C09107=1133.044,378.604,-85.759,-176.914,11.218,149.474
C09108=1133.047,378.356,-85.722,-176.916,11.216,149.474
C09109=1133.051,378.109,-85.685,-176.919,11.213,149.474
C09110=1133.055,377.862,-85.648,-176.921,11.211,149.474
C09111=1133.058,377.615,-85.611,-176.925,11.209,149.474
C09112=1133.062,377.368,-85.574,-176.927,11.207,149.474
C09113=1133.066,377.120,-85.537,-176.930,11.204,149.475
C09114=1133.070,376.874,-85.500,-176.933,11.202,149.475
C09115=1133.073,376.626,-85.463,-176.936,11.200,149.475
C09116=1133.077,376.413,-85.431,-176.938,11.198,149.475
C09117=1133.080,376.200,-85.399,-176.941,11.196,149.475
C09118=1133.084,375.988,-85.367,-176.943,11.194,149.475
C09119=1133.087,375.775,-85.336,-176.945,11.192,149.475
C09120=1133.090,375.562,-85.303,-176.948,11.190,149.475
C09121=1133.093,375.349,-85.272,-176.950,11.188,149.476
C09122=1133.097,375.136,-85.240,-176.953,11.187,149.476
C09123=1133.099,374.924,-85.208,-176.955,11.185,149.476
C09124=1133.104,374.677,-85.171,-176.959,11.182,149.476
C09125=1133.107,374.429,-85.134,-176.962,11.179,149.476
C09126=1133.111,374.182,-85.097,-176.964,11.178,149.476
C09127=1133.114,373.935,-85.061,-176.967,11.175,149.477
C09128=1133.119,373.688,-85.024,-176.970,11.173,149.477
C09129=1133.123,373.440,-84.987,-176.973,11.171,149.477
C09130=1133.126,373.193,-84.950,-176.976,11.168,149.477
C09131=1133.130,372.946,-84.914,-176.979,11.167,149.477
C09132=1133.134,372.699,-84.877,-176.982,11.164,149.477
C09133=1133.138,372.451,-84.840,-176.985,11.161,149.477
C09134=1133.142,372.204,-84.803,-176.988,11.160,149.478
C09135=1133.145,371.957,-84.767,-176.991,11.157,149.478
C09136=1133.149,371.709,-84.730,-176.994,11.155,149.478
C09137=1133.153,371.462,-84.693,-176.997,11.153,149.478
C09138=1133.156,371.215,-84.657,-177.000,11.150,149.478
C09139=1133.160,370.968,-84.620,-177.003,11.148,149.479
C09140=1133.164,370.720,-84.582,-177.006,11.146,149.479
C09141=1133.167,370.473,-84.546,-177.009,11.143,149.479
C09142=1133.171,370.226,-84.510,-177.013,11.141,149.479
C09143=1133.176,369.978,-84.473,-177.015,11.139,149.479
C09144=1133.179,369.731,-84.437,-177.019,11.137,149.480
C09145=1133.183,369.484,-84.400,-177.022,11.134,149.480
C09146=1133.187,369.237,-84.363,-177.025,11.133,149.480
C09147=1133.190,368.989,-84.327,-177.028,11.130,149.480
C09148=1133.194,368.742,-84.290,-177.031,11.128,149.481
C09149=1133.198,368.495,-84.254,-177.034,11.125,149.481
C09150=1133.202,368.248,-84.217,-177.037,11.124,149.481
C09151=1133.206,368.000,-84.180,-177.040,11.121,149.481
C09152=1133.209,367.753,-84.145,-177.044,11.119,149.481
C09153=1133.214,367.506,-84.108,-177.047,11.116,149.482
C09154=1133.217,367.259,-84.072,-177.050,11.114,149.482
C09155=1133.221,367.011,-84.036,-177.053,11.112,149.482
C09156=1133.225,366.764,-83.999,-177.056,11.109,149.482
C09157=1133.229,366.517,-83.963,-177.060,11.107,149.483
C09158=1133.233,366.268,-83.926,-177.063,11.105,149.483
C09159=1133.236,366.022,-83.890,-177.066,11.102,149.483
C09160=1133.240,365.774,-83.853,-177.070,11.100,149.483
C09161=1133.244,365.527,-83.817,-177.072,11.098,149.483
C09162=1133.248,365.280,-83.781,-177.076,11.096,149.484
C09163=1133.251,365.032,-83.745,-177.079,11.093,149.484
C09164=1133.256,364.785,-83.708,-177.083,11.091,149.484
C09165=1133.259,364.537,-83.673,-177.086,11.088,149.484
C09166=1133.263,364.291,-83.636,-177.089,11.086,149.485
C09167=1133.267,364.043,-83.600,-177.092,11.083,149.485
C09168=1133.270,363.796,-83.564,-177.096,11.081,149.485
C09169=1133.275,363.548,-83.528,-177.099,11.079,149.486
C09170=1133.278,363.301,-83.491,-177.102,11.077,149.486
C09171=1133.282,363.054,-83.456,-177.105,11.075,149.486
C09172=1133.286,362.841,-83.424,-177.109,11.072,149.486
C09173=1133.289,362.627,-83.394,-177.111,11.070,149.486
C09174=1133.292,362.415,-83.362,-177.115,11.068,149.487
C09175=1133.295,362.202,-83.331,-177.117,11.066,149.487
C09176=1133.298,361.989,-83.300,-177.120,11.064,149.487
C09177=1133.301,361.776,-83.269,-177.123,11.062,149.487
C09178=1133.305,361.563,-83.239,-177.126,11.060,149.487
C09179=1133.308,361.350,-83.207,-177.129,11.058,149.488
C09180=1133.312,361.102,-83.171,-177.132,11.055,149.488
C09181=1133.316,360.855,-83.136,-177.136,11.053,149.488
C09182=1133.319,360.608,-83.099,-177.139,11.051,149.489
C09183=1133.324,360.360,-83.063,-177.143,11.048,149.489
C09184=1133.327,360.113,-83.028,-177.146,11.046,149.489
C09185=1133.331,359.866,-82.991,-177.150,11.044,149.489
C09186=1133.336,359.619,-82.956,-177.153,11.041,149.490
C09187=1133.339,359.371,-82.920,-177.156,11.039,149.490
C09188=1133.343,359.124,-82.885,-177.160,11.036,149.490
C09189=1133.347,358.876,-82.849,-177.163,11.034,149.490
C09190=1133.351,358.629,-82.812,-177.167,11.032,149.491
C09191=1133.354,358.382,-82.777,-177.170,11.028,149.491
C09192=1133.358,358.134,-82.741,-177.174,11.026,149.491
C09193=1133.362,357.887,-82.705,-177.177,11.024,149.491
C09194=1133.365,357.639,-82.670,-177.181,11.021,149.492
C09195=1133.370,357.391,-82.634,-177.184,11.019,149.492
C09196=1133.374,357.145,-82.599,-177.188,11.017,149.492
C09197=1133.378,356.897,-82.563,-177.191,11.014,149.493
C09198=1133.381,356.650,-82.527,-177.195,11.011,149.493
C09199=1133.385,356.403,-82.491,-177.199,11.009,149.493
C09200=1133.389,356.155,-82.455,-177.202,11.006,149.493
C09201=1133.393,355.907,-82.420,-177.205,11.004,149.494
C09202=1133.396,355.660,-82.384,-177.210,11.001,149.494
C09203=1133.401,355.413,-82.349,-177.213,10.998,149.494
C09204=1133.404,355.166,-82.313,-177.216,10.996,149.494
C09205=1133.408,354.918,-82.278,-177.220,10.994,149.495
C09206=1133.412,354.670,-82.243,-177.224,10.991,149.495
C09207=1133.416,354.422,-82.207,-177.227,10.988,149.495
C09208=1133.420,354.176,-82.172,-177.231,10.986,149.495
C09209=1133.424,353.928,-82.137,-177.234,10.984,149.496
C09210=1133.428,353.680,-82.100,-177.238,10.980,149.496
C09211=1133.432,353.433,-82.065,-177.242,10.978,149.496
C09212=1133.436,353.186,-82.030,-177.245,10.976,149.497
C09213=1133.440,352.938,-81.994,-177.249,10.972,149.497
C09214=1133.444,352.690,-81.959,-177.253,10.970,149.497
C09215=1133.447,352.443,-81.924,-177.256,10.968,149.497
C09216=1133.451,352.195,-81.888,-177.260,10.965,149.498
C09217=1133.455,351.949,-81.853,-177.263,10.962,149.498
C09218=1133.459,351.700,-81.818,-177.267,10.959,149.498
C09219=1133.463,351.453,-81.783,-177.271,10.957,149.498
C09220=1133.467,351.206,-81.748,-177.275,10.954,149.499
C09221=1133.471,350.958,-81.713,-177.278,10.951,149.499
C09222=1133.475,350.711,-81.677,-177.282,10.949,149.499
C09223=1133.478,350.463,-81.642,-177.286,10.946,149.500
C09224=1133.482,350.216,-81.608,-177.289,10.943,149.500
C09225=1133.486,349.968,-81.572,-177.294,10.940,149.500
C09226=1133.489,349.721,-81.537,-177.297,10.938,149.500
C09227=1133.494,349.473,-81.502,-177.301,10.935,149.501
C09228=1133.497,349.260,-81.472,-177.304,10.933,149.501
C09229=1133.501,349.047,-81.441,-177.307,10.930,149.501
C09230=1133.504,348.835,-81.411,-177.309,10.929,149.501
C09231=1133.508,348.621,-81.382,-177.313,10.926,149.501
C09232=1133.511,348.407,-81.351,-177.315,10.924,149.501
C09233=1133.514,348.195,-81.321,-177.317,10.922,149.502
C09234=1133.518,347.982,-81.291,-177.321,10.920,149.502
C09235=1133.521,347.769,-81.260,-177.323,10.918,149.502
C09236=1133.525,347.521,-81.225,-177.326,10.915,149.502
C09237=1133.529,347.273,-81.191,-177.330,10.913,149.502
C09238=1133.532,347.026,-81.156,-177.333,10.911,149.503
C09239=1133.536,346.778,-81.121,-177.336,10.908,149.503
C09240=1133.541,346.531,-81.086,-177.340,10.906,149.503
C09241=1133.545,346.283,-81.051,-177.343,10.903,149.503
C09242=1133.549,346.036,-81.016,-177.346,10.900,149.503
C09243=1133.552,345.788,-80.982,-177.349,10.898,149.504
C09244=1133.557,345.541,-80.947,-177.353,10.895,149.504
C09245=1133.560,345.293,-80.912,-177.356,10.893,149.504
C09246=1133.564,345.045,-80.877,-177.359,10.891,149.504
C09247=1133.568,344.798,-80.843,-177.362,10.888,149.505
C09248=1133.572,344.551,-80.808,-177.366,10.886,149.505
C09249=1133.576,344.303,-80.773,-177.369,10.883,149.505
C09250=1133.580,344.055,-80.739,-177.372,10.880,149.505
C09251=1133.584,343.808,-80.704,-177.375,10.878,149.505
C09252=1133.588,343.560,-80.669,-177.379,10.875,149.506
C09253=1133.592,343.313,-80.634,-177.382,10.873,149.506
C09254=1133.596,343.065,-80.600,-177.385,10.871,149.506
C09255=1133.600,342.817,-80.565,-177.388,10.868,149.506
C09256=1133.604,342.570,-80.531,-177.391,10.865,149.506
C09257=1133.607,342.323,-80.496,-177.395,10.863,149.507
C09258=1133.612,342.075,-80.461,-177.398,10.860,149.507
C09259=1133.616,341.827,-80.427,-177.401,10.858,149.507
C09260=1133.619,341.580,-80.393,-177.405,10.856,149.507
C09261=1133.623,341.332,-80.358,-177.408,10.853,149.507
C09262=1133.627,341.085,-80.324,-177.411,10.850,149.508
C09263=1133.632,340.837,-80.290,-177.414,10.848,149.508
C09264=1133.636,340.589,-80.255,-177.418,10.845,149.508
C09265=1133.640,340.342,-80.221,-177.421,10.843,149.508
C09266=1133.644,340.094,-80.186,-177.424,10.840,149.508
C09267=1133.647,339.847,-80.152,-177.427,10.838,149.509
C09268=1133.651,339.599,-80.117,-177.430,10.835,149.509
C09269=1133.655,339.352,-80.083,-177.434,10.833,149.509
C09270=1133.659,339.103,-80.049,-177.436,10.831,149.509
C09271=1133.663,338.856,-80.015,-177.440,10.829,149.509
C09272=1133.668,338.609,-79.980,-177.443,10.826,149.510
C09273=1133.672,338.361,-79.945,-177.446,10.823,149.510
C09274=1133.675,338.114,-79.912,-177.449,10.821,149.510
C09275=1133.679,337.866,-79.877,-177.453,10.819,149.510
C09276=1133.683,337.618,-79.843,-177.456,10.816,149.510
C09277=1133.686,337.371,-79.809,-177.459,10.813,149.511
C09278=1133.691,337.123,-79.774,-177.462,10.811,149.511
C09279=1133.695,336.875,-79.741,-177.466,10.808,149.511
C09280=1133.699,336.627,-79.706,-177.469,10.806,149.511
C09281=1133.703,336.380,-79.672,-177.472,10.803,149.512
C09282=1133.707,336.132,-79.637,-177.475,10.801,149.512
C09283=1133.711,335.885,-79.604,-177.478,10.798,149.512
C09284=1133.714,335.672,-79.575,-177.482,10.796,149.512
C09285=1133.718,335.458,-79.545,-177.484,10.794,149.512
C09286=1133.721,335.245,-79.516,-177.487,10.792,149.512
C09287=1133.724,335.032,-79.487,-177.490,10.789,149.512
C09288=1133.728,334.819,-79.458,-177.492,10.788,149.513
C09289=1133.731,334.605,-79.428,-177.495,10.785,149.513
C09290=1133.735,334.392,-79.399,-177.498,10.783,149.513
C09291=1133.738,334.178,-79.370,-177.500,10.781,149.513
C09292=1133.743,333.931,-79.335,-177.504,10.779,149.513
C09293=1133.746,333.683,-79.301,-177.507,10.776,149.514
C09294=1133.750,333.436,-79.268,-177.510,10.774,149.514
C09295=1133.754,333.188,-79.233,-177.513,10.771,149.514
C09296=1133.758,332.940,-79.199,-177.516,10.769,149.514
C09297=1133.762,332.693,-79.166,-177.520,10.766,149.514
C09298=1133.766,332.445,-79.132,-177.523,10.764,149.515
C09299=1133.771,332.197,-79.098,-177.526,10.761,149.515
C09300=1133.774,331.950,-79.064,-177.529,10.758,149.515
C09301=1133.778,331.703,-79.030,-177.533,10.756,149.515
C09302=1133.782,331.454,-78.997,-177.536,10.754,149.515
C09303=1133.786,331.207,-78.962,-177.539,10.751,149.515
C09304=1133.790,330.959,-78.929,-177.542,10.748,149.516
C09305=1133.794,330.712,-78.895,-177.546,10.746,149.516
C09306=1133.798,330.464,-78.862,-177.549,10.743,149.516
C09307=1133.802,330.215,-78.828,-177.552,10.741,149.516
C09308=1133.806,329.968,-78.794,-177.555,10.738,149.517
C09309=1133.810,329.721,-78.761,-177.558,10.736,149.517
C09310=1133.814,329.473,-78.727,-177.562,10.733,149.517
C09311=1133.817,329.225,-78.694,-177.565,10.731,149.517
C09312=1133.822,328.978,-78.659,-177.568,10.728,149.517
C09313=1133.826,328.730,-78.626,-177.571,10.726,149.518
C09314=1133.830,328.482,-78.593,-177.574,10.723,149.518
C09315=1133.834,328.235,-78.559,-177.578,10.720,149.518
C09316=1133.838,327.987,-78.525,-177.581,10.718,149.518
C09317=1133.842,327.739,-78.492,-177.584,10.716,149.518
C09318=1133.846,327.492,-78.458,-177.587,10.713,149.518
C09319=1133.850,327.244,-78.425,-177.590,10.710,149.519
C09320=1133.855,326.996,-78.392,-177.594,10.708,149.519
C09321=1133.858,326.748,-78.358,-177.597,10.705,149.519
C09322=1133.862,326.500,-78.324,-177.600,10.703,149.519
C09323=1133.866,326.253,-78.291,-177.603,10.701,149.520
C09324=1133.870,326.005,-78.258,-177.606,10.699,149.520
C09325=1133.874,325.757,-78.225,-177.609,10.696,149.520
C09326=1133.879,325.509,-78.192,-177.612,10.693,149.520
C09327=1133.882,325.262,-78.158,-177.616,10.691,149.520
C09328=1133.886,325.014,-78.124,-177.619,10.688,149.520
C09329=1133.890,324.766,-78.091,-177.622,10.686,149.521
C09330=1133.894,324.518,-78.058,-177.625,10.683,149.521
C09331=1133.898,324.271,-78.025,-177.628,10.680,149.521
C09332=1133.902,324.023,-77.992,-177.631,10.678,149.521
C09333=1133.907,323.775,-77.958,-177.635,10.676,149.521
C09334=1133.911,323.528,-77.925,-177.638,10.673,149.521
C09335=1133.915,323.280,-77.892,-177.641,10.670,149.522
C09336=1133.918,323.031,-77.859,-177.644,10.668,149.522
C09337=1133.922,322.784,-77.825,-177.647,10.665,149.522
C09338=1133.926,322.537,-77.792,-177.651,10.663,149.522
C09339=1133.930,322.289,-77.759,-177.654,10.660,149.523
C09340=1133.934,322.076,-77.731,-177.656,10.658,149.523
C09341=1133.937,321.862,-77.703,-177.660,10.656,149.523
C09342=1133.940,321.649,-77.673,-177.662,10.654,149.523
C09343=1133.944,321.435,-77.645,-177.665,10.651,149.523
C09344=1133.948,321.222,-77.616,-177.667,10.649,149.523
C09345=1133.951,321.008,-77.588,-177.670,10.647,149.523
C09346=1133.955,320.794,-77.560,-177.673,10.645,149.524
C09347=1133.958,320.582,-77.531,-177.675,10.643,149.524
C09348=1133.962,320.334,-77.498,-177.679,10.641,149.524
C09349=1133.966,320.086,-77.466,-177.682,10.638,149.524
C09350=1133.970,319.838,-77.433,-177.685,10.635,149.524
C09351=1133.974,319.590,-77.399,-177.688,10.633,149.525
C09352=1133.978,319.343,-77.367,-177.692,10.630,149.525
C09353=1133.982,319.095,-77.334,-177.695,10.628,149.525
C09354=1133.986,318.847,-77.301,-177.698,10.625,149.525
C09355=1133.991,318.599,-77.268,-177.701,10.622,149.525
C09356=1133.995,318.351,-77.235,-177.704,10.620,149.526
C09357=1133.998,318.104,-77.202,-177.707,10.618,149.526
C09358=1134.002,317.856,-77.169,-177.710,10.615,149.526
C09359=1134.007,317.608,-77.137,-177.714,10.612,149.526
C09360=1134.011,317.360,-77.104,-177.717,10.610,149.526
C09361=1134.014,317.113,-77.071,-177.720,10.607,149.526
C09362=1134.019,316.864,-77.039,-177.723,10.605,149.527
C09363=1134.023,316.617,-77.005,-177.726,10.603,149.527
C09364=1134.026,316.369,-76.973,-177.729,10.600,149.527
C09365=1134.031,316.121,-76.940,-177.732,10.598,149.527
C09366=1134.035,315.873,-76.907,-177.735,10.595,149.527
C09367=1134.038,315.626,-76.875,-177.738,10.593,149.528
C09368=1134.043,315.377,-76.842,-177.742,10.590,149.528
C09369=1134.047,315.130,-76.809,-177.745,10.587,149.528
C09370=1134.050,314.882,-76.777,-177.748,10.585,149.528
C09371=1134.055,314.634,-76.744,-177.751,10.583,149.528
C09372=1134.059,314.387,-76.711,-177.754,10.580,149.529
C09373=1134.063,314.139,-76.680,-177.758,10.577,149.529
C09374=1134.067,313.891,-76.646,-177.761,10.575,149.529
C09375=1134.072,313.643,-76.614,-177.764,10.572,149.529
C09376=1134.075,313.395,-76.581,-177.767,10.570,149.529
C09377=1134.079,313.147,-76.549,-177.770,10.567,149.529
C09378=1134.083,312.899,-76.517,-177.773,10.564,149.530
C09379=1134.087,312.651,-76.484,-177.776,10.562,149.530
C09380=1134.091,312.403,-76.452,-177.780,10.559,149.530
C09381=1134.096,312.156,-76.419,-177.783,10.557,149.530
C09382=1134.100,311.908,-76.387,-177.786,10.554,149.530
C09383=1134.104,311.660,-76.354,-177.789,10.552,149.531
C09384=1134.108,311.412,-76.322,-177.792,10.550,149.531
C09385=1134.112,311.164,-76.290,-177.795,10.547,149.531
C09386=1134.116,310.916,-76.257,-177.798,10.545,149.531
C09387=1134.120,310.669,-76.225,-177.801,10.542,149.531
C09388=1134.125,310.421,-76.193,-177.805,10.540,149.532
C09389=1134.128,310.173,-76.160,-177.807,10.537,149.532
C09390=1134.132,309.925,-76.128,-177.811,10.534,149.532
C09391=1134.136,309.677,-76.096,-177.814,10.532,149.532
C09392=1134.141,309.429,-76.064,-177.817,10.529,149.532
C09393=1134.145,309.182,-76.031,-177.820,10.527,149.533
C09394=1134.148,308.934,-76.000,-177.823,10.524,149.533
C09395=1134.153,308.685,-75.967,-177.827,10.521,149.533
C09396=1134.156,308.472,-75.940,-177.829,10.519,149.533
C09397=1134.160,308.258,-75.912,-177.832,10.517,149.533
C09398=1134.163,308.045,-75.885,-177.835,10.515,149.533
C09399=1134.167,307.831,-75.856,-177.837,10.513,149.533
C09400=1134.170,307.618,-75.829,-177.840,10.511,149.534
C09401=1134.174,307.404,-75.801,-177.843,10.509,149.534
C09402=1134.177,307.191,-75.774,-177.845,10.506,149.534
C09403=1134.181,306.977,-75.746,-177.848,10.504,149.534
C09404=1134.185,306.729,-75.714,-177.851,10.501,149.534
C09405=1134.189,306.481,-75.681,-177.854,10.499,149.535
C09406=1134.194,306.234,-75.650,-177.857,10.496,149.535
C09407=1134.197,305.985,-75.618,-177.861,10.494,149.535
C09408=1134.202,305.737,-75.586,-177.864,10.491,149.535
C09409=1134.206,305.490,-75.554,-177.867,10.489,149.535
C09410=1134.210,305.242,-75.522,-177.870,10.486,149.535
C09411=1134.214,304.993,-75.490,-177.873,10.483,149.536
C09412=1134.218,304.746,-75.458,-177.877,10.481,149.536
C09413=1134.222,304.498,-75.426,-177.879,10.478,149.536
C09414=1134.227,304.250,-75.394,-177.882,10.477,149.536
C09415=1134.230,304.002,-75.362,-177.885,10.474,149.536
C09416=1134.235,303.754,-75.331,-177.888,10.471,149.537
C09417=1134.238,303.506,-75.299,-177.891,10.469,149.537
C09418=1134.243,303.259,-75.267,-177.895,10.466,149.537
C09419=1134.247,303.010,-75.236,-177.898,10.463,149.537
C09420=1134.251,302.762,-75.204,-177.901,10.461,149.537
C09421=1134.255,302.515,-75.172,-177.904,10.459,149.537
C09422=1134.259,302.267,-75.140,-177.907,10.456,149.538
C09423=1134.264,302.018,-75.108,-177.911,10.453,149.538
C09424=1134.268,301.771,-75.077,-177.914,10.451,149.538
C09425=1134.272,301.522,-75.045,-177.917,10.448,149.538
C09426=1134.276,301.275,-75.014,-177.920,10.445,149.538
C09427=1134.280,301.027,-74.982,-177.923,10.443,149.539
C09428=1134.284,300.778,-74.950,-177.926,10.440,149.539
C09429=1134.289,300.531,-74.918,-177.929,10.438,149.539
C09430=1134.293,300.282,-74.887,-177.932,10.436,149.539
C09431=1134.297,300.035,-74.856,-177.935,10.433,149.539
C09432=1134.301,299.787,-74.824,-177.938,10.431,149.539
C09433=1134.305,299.538,-74.793,-177.941,10.428,149.540
C09434=1134.309,299.291,-74.761,-177.944,10.425,149.540
C09435=1134.313,299.043,-74.729,-177.948,10.423,149.540
C09436=1134.317,298.795,-74.699,-177.950,10.420,149.540
C09437=1134.322,298.547,-74.666,-177.954,10.418,149.540
C09438=1134.326,298.299,-74.635,-177.957,10.415,149.540
C09439=1134.330,298.051,-74.603,-177.960,10.413,149.541
C09440=1134.334,297.803,-74.572,-177.963,10.410,149.541
C09441=1134.338,297.555,-74.541,-177.966,10.407,149.541
C09442=1134.342,297.307,-74.509,-177.969,10.405,149.541
C09443=1134.346,297.059,-74.478,-177.973,10.402,149.541
C09444=1134.350,296.811,-74.446,-177.975,10.400,149.542
C09445=1134.355,296.563,-74.415,-177.978,10.398,149.542
C09446=1134.359,296.315,-74.384,-177.981,10.395,149.542
C09447=1134.363,296.067,-74.352,-177.985,10.393,149.542
C09448=1134.367,295.819,-74.321,-177.987,10.390,149.542
C09449=1134.371,295.571,-74.290,-177.991,10.387,149.542
C09450=1134.375,295.323,-74.259,-177.994,10.385,149.543
C09451=1134.380,295.075,-74.228,-177.997,10.382,149.543
C09452=1134.383,294.862,-74.200,-177.999,10.380,149.543
C09453=1134.386,294.648,-74.173,-178.002,10.377,149.543
C09454=1134.390,294.434,-74.147,-178.005,10.376,149.543
C09455=1134.393,294.220,-74.120,-178.008,10.373,149.543
C09456=1134.397,294.007,-74.093,-178.010,10.371,149.544
C09457=1134.401,293.793,-74.066,-178.013,10.369,149.544
C09458=1134.404,293.579,-74.039,-178.016,10.367,149.544
C09459=1134.408,293.365,-74.013,-178.018,10.365,149.544
C09460=1134.412,293.118,-73.982,-178.022,10.362,149.544
C09461=1134.416,292.869,-73.951,-178.024,10.359,149.544
C09462=1134.421,292.621,-73.920,-178.028,10.357,149.545
C09463=1134.424,292.373,-73.888,-178.031,10.354,149.545
C09464=1134.428,292.125,-73.858,-178.034,10.352,149.545
C09465=1134.433,291.877,-73.827,-178.037,10.349,149.545
C09466=1134.437,291.629,-73.795,-178.040,10.346,149.545
C09467=1134.441,291.381,-73.765,-178.043,10.345,149.546
C09468=1134.445,291.133,-73.733,-178.046,10.342,149.546
C09469=1134.449,290.885,-73.703,-178.049,10.340,149.546
C09470=1134.454,290.637,-73.672,-178.052,10.337,149.546
C09471=1134.457,290.389,-73.641,-178.055,10.334,149.546
C09472=1134.462,290.141,-73.610,-178.058,10.332,149.546
C09473=1134.466,289.892,-73.579,-178.062,10.329,149.547
C09474=1134.470,289.645,-73.549,-178.064,10.326,149.547
C09475=1134.474,289.397,-73.518,-178.068,10.324,149.547
C09476=1134.479,289.148,-73.487,-178.071,10.321,149.547
C09477=1134.482,288.900,-73.457,-178.074,10.319,149.547
C09478=1134.487,288.653,-73.426,-178.077,10.316,149.547
C09479=1134.491,288.404,-73.395,-178.080,10.314,149.548
C09480=1134.496,288.156,-73.364,-178.083,10.312,149.548
C09481=1134.499,287.909,-73.333,-178.086,10.309,149.548
C09482=1134.503,287.660,-73.302,-178.089,10.306,149.548
C09483=1134.508,287.412,-73.271,-178.092,10.304,149.548
C09484=1134.512,287.165,-73.241,-178.095,10.301,149.549
C09485=1134.516,286.916,-73.210,-178.098,10.298,149.549
C09486=1134.521,286.667,-73.180,-178.101,10.296,149.549
C09487=1134.524,286.420,-73.150,-178.104,10.293,149.549
C09488=1134.529,286.171,-73.118,-178.108,10.291,149.549
C09489=1134.532,285.923,-73.088,-178.111,10.288,149.549
C09490=1134.537,285.675,-73.058,-178.114,10.285,149.550
C09491=1134.542,285.428,-73.027,-178.116,10.284,149.550
C09492=1134.545,285.179,-72.996,-178.119,10.281,149.550
C09493=1134.549,284.931,-72.965,-178.123,10.279,149.550
C09494=1134.553,284.684,-72.935,-178.126,10.276,149.550
C09495=1134.558,284.436,-72.905,-178.129,10.273,149.551
C09496=1134.562,284.186,-72.874,-178.132,10.271,149.551
C09497=1134.566,283.939,-72.844,-178.135,10.268,149.551
C09498=1134.571,283.691,-72.813,-178.138,10.265,149.551
C09499=1134.575,283.443,-72.783,-178.141,10.263,149.551
C09500=1134.579,283.194,-72.752,-178.144,10.260,149.551
C09501=1134.583,282.946,-72.722,-178.147,10.257,149.552
C09502=1134.587,282.698,-72.692,-178.150,10.256,149.552
C09503=1134.591,282.451,-72.661,-178.153,10.253,149.552
C09504=1134.596,282.202,-72.631,-178.156,10.251,149.552
C09505=1134.600,281.954,-72.601,-178.159,10.248,149.552
C09506=1134.604,281.706,-72.570,-178.162,10.245,149.552
C09507=1134.608,281.458,-72.540,-178.166,10.243,149.553
C09508=1134.612,281.244,-72.514,-178.168,10.240,149.553
C09509=1134.616,281.030,-72.488,-178.172,10.238,149.553
C09510=1134.619,280.816,-72.462,-178.175,10.235,149.553
C09511=1134.623,280.603,-72.436,-178.178,10.232,149.553
C09512=1134.627,280.388,-72.410,-178.181,10.230,149.554
C09513=1134.630,280.175,-72.385,-178.184,10.227,149.554
C09514=1134.634,279.961,-72.358,-178.188,10.225,149.554
C09515=1134.637,279.746,-72.332,-178.191,10.222,149.554
C09516=1134.642,279.498,-72.302,-178.194,10.220,149.555
C09517=1134.646,279.250,-72.271,-178.198,10.216,149.555
C09518=1134.650,279.003,-72.241,-178.201,10.214,149.555
C09519=1134.654,278.754,-72.212,-178.205,10.211,149.555
C09520=1134.659,278.506,-72.182,-178.208,10.208,149.555
C09521=1134.663,278.258,-72.152,-178.212,10.206,149.556
C09522=1134.667,278.009,-72.122,-178.215,10.202,149.556
C09523=1134.670,277.761,-72.092,-178.219,10.200,149.556
C09524=1134.675,277.513,-72.062,-178.222,10.196,149.556
C09525=1134.679,277.265,-72.031,-178.225,10.194,149.556
C09526=1134.683,277.017,-72.002,-178.228,10.191,149.557
C09527=1134.688,276.768,-71.972,-178.232,10.188,149.557
C09528=1134.692,276.521,-71.942,-178.235,10.185,149.557
C09529=1134.696,276.272,-71.912,-178.239,10.183,149.557
C09530=1134.701,276.024,-71.883,-178.242,10.180,149.557
C09531=1134.704,275.777,-71.853,-178.245,10.176,149.557
C09532=1134.709,275.528,-71.823,-178.249,10.174,149.558
C09533=1134.714,275.280,-71.793,-178.251,10.171,149.558
C09534=1134.717,275.032,-71.763,-178.254,10.168,149.558
C09535=1134.722,274.784,-71.734,-178.258,10.166,149.558
C09536=1134.726,274.536,-71.704,-178.261,10.163,149.558
C09537=1134.731,274.287,-71.674,-178.264,10.160,149.558
C09538=1134.735,274.039,-71.644,-178.267,10.157,149.558
C09539=1134.739,273.791,-71.614,-178.271,10.155,149.559
C09540=1134.743,273.543,-71.585,-178.274,10.152,149.559
C09541=1134.747,273.295,-71.556,-178.276,10.149,149.559
C09542=1134.751,273.046,-71.526,-178.279,10.146,149.559
C09543=1134.756,272.798,-71.497,-178.282,10.144,149.559
C09544=1134.760,272.550,-71.466,-178.285,10.141,149.559
C09545=1134.764,272.302,-71.436,-178.289,10.138,149.560
C09546=1134.769,272.053,-71.407,-178.291,10.136,149.560
C09547=1134.773,271.805,-71.377,-178.294,10.134,149.560
C09548=1134.777,271.557,-71.348,-178.297,10.131,149.560
C09549=1134.781,271.309,-71.319,-178.300,10.128,149.560
C09550=1134.785,271.060,-71.289,-178.303,10.125,149.560
C09551=1134.789,270.812,-71.260,-178.306,10.123,149.560
C09552=1134.794,270.564,-71.230,-178.308,10.121,149.560
C09553=1134.798,270.316,-71.201,-178.311,10.118,149.560
C09554=1134.802,270.067,-71.171,-178.314,10.115,149.561
C09555=1134.806,269.819,-71.142,-178.317,10.112,149.561
C09556=1134.810,269.571,-71.112,-178.319,10.110,149.561
C09557=1134.815,269.323,-71.083,-178.322,10.108,149.561
C09558=1134.819,269.075,-71.054,-178.325,10.105,149.561
C09559=1134.823,268.827,-71.024,-178.327,10.103,149.561
C09560=1134.828,268.578,-70.995,-178.330,10.100,149.561
C09561=1134.832,268.330,-70.966,-178.332,10.098,149.561
C09562=1134.836,268.082,-70.936,-178.335,10.095,149.561
C09563=1134.840,267.833,-70.907,-178.337,10.093,149.561
C09564=1134.844,267.620,-70.882,-178.340,10.091,149.561
C09565=1134.848,267.405,-70.856,-178.342,10.089,149.562
C09566=1134.852,267.191,-70.832,-178.344,10.087,149.562
C09567=1134.855,266.978,-70.806,-178.346,10.085,149.562
C09568=1134.859,266.763,-70.781,-178.348,10.083,149.562
C09569=1134.863,266.549,-70.756,-178.351,10.081,149.562
C09570=1134.866,266.336,-70.731,-178.353,10.079,149.562
C09571=1134.870,266.121,-70.706,-178.355,10.077,149.562
C09572=1134.874,265.873,-70.676,-178.357,10.075,149.562
C09573=1134.879,265.625,-70.647,-178.360,10.071,149.562
C09574=1134.883,265.377,-70.618,-178.362,10.069,149.562
C09575=1134.887,265.128,-70.589,-178.364,10.067,149.562
C09576=1134.891,264.880,-70.560,-178.367,10.065,149.562
C09577=1134.896,264.631,-70.530,-178.370,10.063,149.563
C09578=1134.900,264.384,-70.502,-178.372,10.061,149.563
C09579=1134.904,264.135,-70.473,-178.376,10.058,149.563
C09580=1134.908,263.887,-70.443,-178.381,10.054,149.563
C09581=1134.913,263.639,-70.414,-178.385,10.050,149.563
C09582=1134.917,263.390,-70.385,-178.389,10.047,149.564
C09583=1134.922,263.142,-70.356,-178.393,10.044,149.564
C09584=1134.926,262.894,-70.328,-178.396,10.041,149.564
C09585=1134.930,262.646,-70.299,-178.400,10.037,149.564
C09586=1134.934,262.397,-70.269,-178.404,10.034,149.565
C09587=1134.939,262.149,-70.241,-178.408,10.031,149.565
C09588=1134.942,261.901,-70.212,-178.412,10.028,149.565
C09589=1134.947,261.652,-70.183,-178.416,10.024,149.565
C09590=1134.951,261.404,-70.154,-178.420,10.021,149.566
C09591=1134.956,261.156,-70.125,-178.423,10.018,149.566
C09592=1134.960,260.908,-70.096,-178.427,10.015,149.566
C09593=1134.964,260.659,-70.068,-178.430,10.012,149.566
C09594=1134.969,260.411,-70.039,-178.434,10.009,149.566
C09595=1134.973,260.163,-70.010,-178.437,10.006,149.566
C09596=1134.977,259.914,-69.982,-178.441,10.003,149.567
C09597=1134.981,259.667,-69.953,-178.445,9.999,149.567
C09598=1134.986,259.418,-69.924,-178.448,9.996,149.567
C09599=1134.990,259.169,-69.896,-178.451,9.993,149.567
C09600=1134.994,258.921,-69.867,-178.455,9.990,149.567
C09601=1134.999,258.673,-69.839,-178.458,9.987,149.567
C09602=1135.003,258.424,-69.810,-178.461,9.984,149.568
C09603=1135.007,258.177,-69.781,-178.465,9.981,149.568
C09604=1135.012,257.928,-69.753,-178.468,9.978,149.568
C09605=1135.015,257.679,-69.724,-178.470,9.975,149.568
C09606=1135.020,257.432,-69.695,-178.473,9.972,149.568
C09607=1135.024,257.183,-69.667,-178.477,9.969,149.568
C09608=1135.028,256.934,-69.638,-178.480,9.966,149.568
C09609=1135.033,256.686,-69.611,-178.483,9.963,149.568
C09610=1135.037,256.437,-69.582,-178.486,9.961,149.568
C09611=1135.041,256.190,-69.553,-178.489,9.958,149.569
C09612=1135.046,255.941,-69.525,-178.491,9.955,149.568
C09613=1135.050,255.693,-69.497,-178.490,9.954,149.568
C09614=1135.055,255.444,-69.468,-178.489,9.954,149.568
C09615=1135.058,255.196,-69.440,-178.488,9.954,149.567
C09616=1135.064,254.948,-69.412,-178.487,9.953,149.567
C09617=1135.067,254.700,-69.383,-178.486,9.953,149.567
C09618=1135.071,254.451,-69.354,-178.486,9.951,149.566
C09619=1135.076,254.203,-69.326,-178.486,9.950,149.566
C09620=1135.082,253.851,-69.286,-178.487,9.950,149.566
C09621=1135.089,253.497,-69.246,-178.488,9.947,149.566
C09622=1135.107,252.397,-69.120,-177.589,8.141,148.878
C09623=1135.111,252.177,-69.096,-177.592,8.138,148.879
C09624=1135.115,251.958,-69.071,-177.594,8.136,148.879
C09625=1135.119,251.738,-69.046,-177.597,8.133,148.879
C09626=1135.123,251.489,-69.018,-177.599,8.130,148.879
C09627=1135.128,251.241,-68.991,-177.602,8.127,148.879
C09628=1135.132,250.992,-68.963,-177.605,8.124,148.879
C09629=1135.136,250.744,-68.935,-177.608,8.121,148.879
C09630=1135.141,250.496,-68.908,-177.610,8.118,148.879
C09631=1135.145,250.247,-68.880,-177.614,8.114,148.879
C09632=1135.150,249.998,-68.852,-177.616,8.111,148.879
C09633=1135.154,249.751,-68.825,-177.619,8.108,148.879
C09634=1135.158,249.502,-68.797,-177.622,8.105,148.879
C09635=1135.162,249.254,-68.769,-177.624,8.102,148.879
C09636=1135.166,249.005,-68.741,-177.627,8.099,148.879
C09637=1135.171,248.756,-68.714,-177.630,8.096,148.879
C09638=1135.175,248.509,-68.687,-177.633,8.093,148.879
C09639=1135.180,248.260,-68.659,-177.636,8.091,148.879
C09640=1135.184,248.011,-68.631,-177.638,8.088,148.879
C09641=1135.189,247.763,-68.604,-177.641,8.084,148.879
C09642=1135.193,247.515,-68.576,-177.644,8.082,148.879
C09643=1135.197,247.266,-68.548,-177.647,8.078,148.879
C09644=1135.202,247.017,-68.521,-177.650,8.075,148.879
C09645=1135.206,246.769,-68.494,-177.653,8.072,148.880
C09646=1135.210,246.520,-68.466,-177.655,8.069,148.880
C09647=1135.215,246.272,-68.438,-177.658,8.066,148.880
C09648=1135.219,246.024,-68.411,-177.661,8.063,148.880
C09649=1135.224,245.775,-68.384,-177.664,8.060,148.880
C09650=1135.228,245.527,-68.356,-177.667,8.057,148.880
C09651=1135.233,245.278,-68.329,-177.669,8.054,148.880
C09652=1135.237,245.030,-68.302,-177.672,8.051,148.880
C09653=1135.242,244.781,-68.275,-177.675,8.048,148.880
C09654=1135.245,244.533,-68.247,-177.677,8.045,148.880
C09655=1135.250,244.284,-68.220,-177.680,8.043,148.880
C09656=1135.254,244.036,-68.193,-177.683,8.040,148.880
C09657=1135.259,243.788,-68.166,-177.686,8.037,148.880
C09658=1135.263,243.539,-68.138,-177.689,8.034,148.880
C09659=1135.267,243.290,-68.111,-177.691,8.031,148.880
C09660=1135.272,243.042,-68.084,-177.694,8.028,148.880
C09661=1135.277,242.793,-68.057,-177.698,8.024,148.881
C09662=1135.281,242.545,-68.029,-177.700,8.021,148.881
C09663=1135.284,242.297,-68.002,-177.703,8.018,148.881
C09664=1135.289,242.048,-67.975,-177.706,8.016,148.881
C09665=1135.294,241.800,-67.948,-177.708,8.012,148.881
C09666=1135.298,241.551,-67.921,-177.711,8.009,148.881
C09667=1135.303,241.303,-67.894,-177.714,8.006,148.881
C09668=1135.308,241.054,-67.867,-177.717,8.004,148.881
C09669=1135.311,240.805,-67.840,-177.720,8.001,148.881
C09670=1135.315,240.557,-67.813,-177.722,7.998,148.881
C09671=1135.320,240.308,-67.786,-177.725,7.995,148.881
C09672=1135.325,240.060,-67.759,-177.728,7.992,148.881
C09673=1135.328,239.812,-67.732,-177.731,7.989,148.881
C09674=1135.333,239.564,-67.705,-177.734,7.986,148.881
C09675=1135.338,239.315,-67.678,-177.736,7.983,148.881
C09676=1135.343,239.066,-67.651,-177.739,7.980,148.882
C09677=1135.346,238.817,-67.624,-177.742,7.977,148.882
C09678=1135.351,238.569,-67.597,-177.745,7.975,148.882
C09679=1135.355,238.320,-67.570,-177.748,7.972,148.882
C09680=1135.360,238.072,-67.543,-177.750,7.969,148.882
C09681=1135.364,237.823,-67.517,-177.753,7.966,148.882
C09682=1135.369,237.575,-67.490,-177.756,7.963,148.882
C09683=1135.373,237.326,-67.463,-177.759,7.960,148.882
C09684=1135.377,237.078,-67.436,-177.762,7.957,148.882
C09685=1135.382,236.830,-67.409,-177.764,7.954,148.882
C09686=1135.386,236.581,-67.382,-177.767,7.951,148.882
C09687=1135.391,236.333,-67.356,-177.770,7.948,148.882
C09688=1135.395,236.084,-67.329,-177.773,7.945,148.882
C09689=1135.400,235.836,-67.302,-177.776,7.943,148.883
C09690=1135.404,235.564,-67.273,-177.778,7.940,148.883
C09691=1135.409,235.291,-67.244,-177.782,7.936,148.883
C09692=1135.414,235.019,-67.215,-177.785,7.933,148.883
C09693=1135.419,234.747,-67.185,-177.788,7.930,148.883
C09694=1135.423,234.499,-67.159,-177.790,7.927,148.883
C09695=1135.428,234.250,-67.133,-177.793,7.924,148.883
C09696=1135.432,234.002,-67.106,-177.796,7.921,148.883
C09697=1135.436,233.753,-67.079,-177.799,7.918,148.883
C09698=1135.441,233.505,-67.053,-177.802,7.916,148.883
C09699=1135.445,233.256,-67.026,-177.804,7.913,148.883
C09700=1135.450,233.008,-66.999,-177.807,7.910,148.883
C09701=1135.454,232.759,-66.973,-177.810,7.907,148.884
C09702=1135.459,232.510,-66.946,-177.813,7.904,148.884
C09703=1135.463,232.262,-66.920,-177.816,7.901,148.884
C09704=1135.467,232.013,-66.894,-177.819,7.898,148.884
C09705=1135.472,231.765,-66.867,-177.822,7.896,148.884
C09706=1135.476,231.516,-66.841,-177.824,7.893,148.884
C09707=1135.480,231.268,-66.814,-177.827,7.890,148.884
C09708=1135.485,231.019,-66.789,-177.830,7.887,148.884
C09709=1135.489,230.770,-66.761,-177.833,7.884,148.884
C09710=1135.494,230.522,-66.736,-177.836,7.881,148.885
C09711=1135.499,230.274,-66.709,-177.838,7.878,148.885
C09712=1135.503,230.025,-66.683,-177.841,7.875,148.885
C09713=1135.507,229.777,-66.657,-177.844,7.872,148.885
C09714=1135.512,229.528,-66.630,-177.847,7.869,148.885
C09715=1135.516,229.279,-66.604,-177.850,7.867,148.885
C09716=1135.521,229.030,-66.578,-177.853,7.864,148.885
C09717=1135.525,228.782,-66.551,-177.855,7.861,148.885
C09718=1135.529,228.533,-66.525,-177.858,7.859,148.885
C09719=1135.534,228.284,-66.499,-177.860,7.856,148.885
C09720=1135.538,228.037,-66.473,-177.863,7.853,148.885
C09721=1135.543,227.788,-66.447,-177.866,7.850,148.886
C09722=1135.547,227.539,-66.420,-177.869,7.847,148.886
C09723=1135.551,227.291,-66.394,-177.872,7.844,148.886
C09724=1135.556,227.042,-66.369,-177.875,7.842,148.886
C09725=1135.560,226.793,-66.342,-177.878,7.839,148.886
C09726=1135.565,226.544,-66.316,-177.880,7.836,148.886
C09727=1135.569,226.296,-66.290,-177.883,7.833,148.886
C09728=1135.574,226.048,-66.265,-177.886,7.830,148.886
C09729=1135.578,225.799,-66.238,-177.889,7.827,148.887
C09730=1135.583,225.550,-66.212,-177.892,7.824,148.887
C09731=1135.587,225.301,-66.186,-177.895,7.821,148.887
C09732=1135.592,225.053,-66.160,-177.898,7.819,148.887
C09733=1135.596,224.805,-66.134,-177.900,7.817,148.887
C09734=1135.600,224.556,-66.108,-177.903,7.814,148.887
C09735=1135.605,224.307,-66.082,-177.906,7.811,148.887
C09736=1135.609,224.058,-66.056,-177.908,7.808,148.887
C09737=1135.614,223.810,-66.030,-177.911,7.805,148.888
C09738=1135.619,223.561,-66.005,-177.914,7.802,148.888
C09739=1135.623,223.312,-65.979,-177.917,7.799,148.888
C09740=1135.627,223.064,-65.953,-177.920,7.796,148.888
C09741=1135.632,222.816,-65.927,-177.923,7.794,148.888
C09742=1135.636,222.567,-65.901,-177.926,7.791,148.888
C09743=1135.641,222.318,-65.875,-177.928,7.789,148.888
C09744=1135.645,222.069,-65.849,-177.931,7.786,148.888
C09745=1135.650,221.821,-65.824,-177.934,7.783,148.889
C09746=1135.654,221.572,-65.798,-177.936,7.780,148.889
C09747=1135.658,221.324,-65.772,-177.939,7.777,148.889
C09748=1135.663,221.075,-65.747,-177.942,7.775,148.889
C09749=1135.667,220.827,-65.721,-177.945,7.772,148.889
C09750=1135.672,220.578,-65.696,-177.948,7.769,148.889
C09751=1135.676,220.329,-65.670,-177.951,7.766,148.889
C09752=1135.681,220.081,-65.644,-177.953,7.764,148.889
C09753=1135.686,219.832,-65.618,-177.956,7.761,148.890
C09754=1135.690,219.583,-65.592,-177.959,7.758,148.890
C09755=1135.695,219.335,-65.567,-177.962,7.755,148.890
C09756=1135.699,219.086,-65.542,-177.965,7.752,148.890
C09757=1135.703,218.837,-65.516,-177.968,7.750,148.890
C09758=1135.708,218.589,-65.491,-177.970,7.747,148.890
C09759=1135.713,218.340,-65.465,-177.973,7.744,148.890
C09760=1135.717,218.091,-65.439,-177.976,7.742,148.891
C09761=1135.722,217.843,-65.414,-177.979,7.739,148.891
C09762=1135.726,217.594,-65.388,-177.982,7.736,148.891
C09763=1135.730,217.345,-65.364,-177.984,7.733,148.891
C09764=1135.734,217.097,-65.338,-177.987,7.730,148.891
C09765=1135.739,216.848,-65.313,-177.990,7.728,148.891
C09766=1135.743,216.599,-65.287,-177.993,7.725,148.891
C09767=1135.748,216.351,-65.262,-177.996,7.723,148.892
C09768=1135.752,216.102,-65.236,-177.998,7.720,148.892
C09769=1135.757,215.854,-65.211,-178.001,7.717,148.892
C09770=1135.761,215.605,-65.185,-178.004,7.714,148.892
C09771=1135.766,215.355,-65.160,-178.007,7.712,148.892
C09772=1135.771,215.107,-65.135,-178.010,7.709,148.892
C09773=1135.775,214.859,-65.109,-178.013,7.706,148.892
C09774=1135.779,214.610,-65.085,-178.015,7.704,148.893
C09775=1135.783,214.361,-65.059,-178.018,7.701,148.893
C09776=1135.788,214.113,-65.034,-178.021,7.698,148.893
C09777=1135.793,213.864,-65.009,-178.024,7.695,148.893
C09778=1135.797,213.615,-64.983,-178.027,7.693,148.893
C09779=1135.802,213.366,-64.958,-178.030,7.690,148.893
C09780=1135.806,213.117,-64.933,-178.032,7.688,148.894
C09781=1135.810,212.870,-64.908,-178.035,7.685,148.894
C09782=1135.815,212.620,-64.883,-178.038,7.682,148.894
C09783=1135.820,212.372,-64.857,-178.041,7.679,148.894
C09784=1135.824,212.123,-64.832,-178.044,7.677,148.894
C09785=1135.828,211.875,-64.808,-178.047,7.674,148.894
C09786=1135.833,211.626,-64.783,-178.049,7.672,148.894
C09787=1135.838,211.377,-64.757,-178.052,7.669,148.895
C09788=1135.842,211.128,-64.732,-178.055,7.666,148.895
C09789=1135.846,210.880,-64.707,-178.058,7.663,148.895
C09790=1135.851,210.631,-64.682,-178.061,7.660,148.895
C09791=1135.856,210.382,-64.658,-178.063,7.658,148.895
C09792=1135.860,210.133,-64.632,-178.066,7.656,148.896
C09793=1135.865,209.885,-64.608,-178.069,7.653,148.896
C09794=1135.870,209.614,-64.580,-178.072,7.650,148.896
C09795=1135.875,209.343,-64.553,-178.075,7.647,148.896
C09796=1135.880,209.073,-64.526,-178.078,7.645,148.896
C09797=1135.884,208.802,-64.499,-178.081,7.641,148.896
C09798=1135.889,208.554,-64.474,-178.084,7.639,148.897
C09799=1135.894,208.304,-64.449,-178.087,7.636,148.897
C09800=1135.898,208.056,-64.425,-178.090,7.633,148.897
C09801=1135.903,207.808,-64.399,-178.093,7.631,148.897
C09802=1135.907,207.559,-64.375,-178.095,7.629,148.897
C09803=1135.912,207.310,-64.350,-178.098,7.626,148.897
C09804=1135.916,207.061,-64.325,-178.101,7.623,148.898
C09805=1135.920,206.813,-64.300,-178.104,7.620,148.898
C09806=1135.925,206.563,-64.275,-178.107,7.617,148.898
C09807=1135.929,206.315,-64.251,-178.109,7.615,148.898
C09808=1135.934,206.066,-64.227,-178.112,7.613,148.898
C09809=1135.939,205.817,-64.201,-178.115,7.610,148.898
C09810=1135.943,205.569,-64.177,-178.118,7.607,148.899
C09811=1135.948,205.320,-64.152,-178.121,7.605,148.899
C09812=1135.952,205.071,-64.128,-178.124,7.602,148.899
C09813=1135.957,204.822,-64.103,-178.126,7.599,148.899
C09814=1135.962,204.574,-64.079,-178.130,7.597,148.899
C09815=1135.966,204.324,-64.054,-178.132,7.594,148.900
C09816=1135.970,204.077,-64.029,-178.135,7.592,148.900
C09817=1135.975,203.828,-64.005,-178.138,7.589,148.900
C09818=1135.979,203.579,-63.980,-178.141,7.586,148.900
C09819=1135.984,203.330,-63.955,-178.144,7.584,148.900
C09820=1135.989,203.082,-63.931,-178.146,7.582,148.901
C09821=1135.993,202.832,-63.906,-178.149,7.579,148.901
C09822=1135.998,202.584,-63.882,-178.152,7.576,148.901
C09823=1136.003,202.335,-63.858,-178.155,7.574,148.901
C09824=1136.006,202.086,-63.833,-178.157,7.571,148.901
C09825=1136.012,201.837,-63.808,-178.160,7.569,148.901
C09826=1136.016,201.589,-63.784,-178.163,7.566,148.902
C09827=1136.020,201.340,-63.760,-178.166,7.564,148.902
C09828=1136.025,201.091,-63.735,-178.169,7.561,148.902
C09829=1136.029,200.843,-63.711,-178.172,7.558,148.902
C09830=1136.034,200.594,-63.687,-178.175,7.556,148.902
C09831=1136.039,200.344,-63.663,-178.177,7.554,148.903
C09832=1136.043,200.096,-63.639,-178.180,7.551,148.903
C09833=1136.048,199.847,-63.614,-178.183,7.548,148.903
C09834=1136.052,199.599,-63.590,-178.186,7.545,148.903
C09835=1136.056,199.350,-63.566,-178.188,7.543,148.903
C09836=1136.061,199.101,-63.541,-178.191,7.541,148.904
C09837=1136.066,198.852,-63.517,-178.195,7.538,148.904
C09838=1136.070,198.603,-63.493,-178.197,7.536,148.904
C09839=1136.075,198.354,-63.468,-178.200,7.533,148.904
C09840=1136.079,198.106,-63.444,-178.203,7.530,148.904
C09841=1136.084,197.857,-63.420,-178.205,7.528,148.905
C09842=1136.088,197.609,-63.396,-178.208,7.526,148.905
C09843=1136.094,197.359,-63.372,-178.211,7.523,148.905
C09844=1136.097,197.110,-63.348,-178.214,7.520,148.905
C09845=1136.102,196.862,-63.324,-178.217,7.518,148.905
C09846=1136.106,196.613,-63.300,-178.220,7.515,148.906
C09847=1136.112,196.364,-63.276,-178.223,7.513,148.906
C09848=1136.116,196.116,-63.252,-178.225,7.511,148.906
C09849=1136.120,195.867,-63.227,-178.228,7.508,148.906
C09850=1136.125,195.617,-63.204,-178.231,7.505,148.906
C09851=1136.130,195.369,-63.179,-178.233,7.503,148.907
C09852=1136.134,195.120,-63.156,-178.237,7.501,148.907
C09853=1136.139,194.871,-63.132,-178.239,7.498,148.907
C09854=1136.143,194.623,-63.108,-178.242,7.496,148.907
C09855=1136.148,194.374,-63.084,-178.245,7.493,148.908
C09856=1136.152,194.125,-63.060,-178.248,7.491,148.908
C09857=1136.157,193.875,-63.036,-178.250,7.489,148.908
C09858=1136.161,193.627,-63.012,-178.253,7.486,148.908
C09859=1136.166,193.379,-62.988,-178.257,7.483,148.908
C09860=1136.171,193.130,-62.964,-178.259,7.481,148.909
C09861=1136.175,192.881,-62.940,-178.262,7.479,148.909
C09862=1136.180,192.632,-62.917,-178.265,7.476,148.909
C09863=1136.184,192.384,-62.893,-178.268,7.474,148.909
C09864=1136.189,192.135,-62.869,-178.270,7.471,148.910
C09865=1136.194,191.886,-62.845,-178.274,7.468,148.910
C09866=1136.198,191.636,-62.821,-178.276,7.466,148.910
C09867=1136.203,191.387,-62.798,-178.279,7.464,148.910
C09868=1136.207,191.139,-62.774,-178.282,7.461,148.910
C09869=1136.212,190.890,-62.750,-178.284,7.459,148.911
C09870=1136.216,190.641,-62.726,-178.288,7.456,148.911
C09871=1136.221,190.392,-62.703,-178.290,7.453,148.911
C09872=1136.226,190.143,-62.680,-178.293,7.452,148.911
C09873=1136.230,189.895,-62.655,-178.296,7.449,148.912
C09874=1136.235,189.646,-62.632,-178.299,7.446,148.912
C09875=1136.239,189.397,-62.609,-178.301,7.444,148.912
C09876=1136.244,189.148,-62.585,-178.305,7.442,148.912
C09877=1136.248,188.899,-62.561,-178.308,7.439,148.912
C09878=1136.253,188.650,-62.538,-178.310,7.437,148.913
C09879=1136.258,188.402,-62.514,-178.313,7.434,148.913
C09880=1136.262,188.153,-62.490,-178.316,7.432,148.913
C09881=1136.267,187.904,-62.467,-178.319,7.430,148.913
C09882=1136.272,187.655,-62.444,-178.322,7.427,148.914
C09883=1136.276,187.406,-62.420,-178.324,7.425,148.914
C09884=1136.281,187.157,-62.396,-178.327,7.422,148.914
C09885=1136.285,186.908,-62.373,-178.330,7.420,148.914
C09886=1136.289,186.660,-62.350,-178.333,7.418,148.915
C09887=1136.294,186.411,-62.326,-178.336,7.415,148.915
C09888=1136.298,186.162,-62.303,-178.338,7.413,148.915
C09889=1136.303,185.913,-62.279,-178.341,7.410,148.915
C09890=1136.308,185.664,-62.256,-178.345,7.408,148.916
C09891=1136.313,185.415,-62.233,-178.347,7.406,148.916
C09892=1136.318,185.167,-62.210,-178.350,7.403,148.916
C09893=1136.323,184.918,-62.186,-178.352,7.401,148.916
C09894=1136.327,184.669,-62.164,-178.356,7.399,148.917
C09895=1136.331,184.421,-62.140,-178.358,7.396,148.917
C09896=1136.336,184.172,-62.116,-178.361,7.394,148.917
C09897=1136.340,183.923,-62.093,-178.364,7.391,148.917
C09898=1136.346,183.653,-62.068,-178.367,7.388,148.918
C09899=1136.351,183.383,-62.043,-178.370,7.387,148.918
C09900=1136.355,183.113,-62.018,-178.373,7.384,148.918
C09901=1136.360,182.844,-61.992,-178.376,7.381,148.918
C09902=1136.365,182.595,-61.969,-178.379,7.379,148.919
C09903=1136.369,182.346,-61.945,-178.382,7.377,148.919
C09904=1136.374,182.098,-61.923,-178.385,7.374,148.919
C09905=1136.379,181.849,-61.900,-178.388,7.371,148.919
C09906=1136.383,181.600,-61.876,-178.390,7.370,148.920
C09907=1136.388,181.350,-61.854,-178.393,7.367,148.920
C09908=1136.392,181.101,-61.831,-178.396,7.365,148.920
C09909=1136.397,180.852,-61.808,-178.399,7.362,148.920
C09910=1136.402,180.603,-61.784,-178.401,7.360,148.921
C09911=1136.406,180.355,-61.762,-178.405,7.358,148.921
C09912=1136.411,180.106,-61.738,-178.407,7.355,148.921
C09913=1136.416,179.857,-61.715,-178.410,7.353,148.922
C09914=1136.420,179.608,-61.692,-178.413,7.350,148.922
C09915=1136.425,179.359,-61.670,-178.416,7.349,148.922
C09916=1136.430,179.110,-61.647,-178.419,7.346,148.922
C09917=1136.434,178.862,-61.624,-178.421,7.344,148.923
C09918=1136.439,178.613,-61.601,-178.425,7.341,148.923
C09919=1136.443,178.364,-61.577,-178.427,7.339,148.923
C09920=1136.448,178.114,-61.555,-178.430,7.337,148.923
C09921=1136.453,177.866,-61.532,-178.432,7.335,148.924
C09922=1136.457,177.617,-61.509,-178.436,7.332,148.924
C09923=1136.462,177.368,-61.486,-178.438,7.329,148.924
C09924=1136.467,177.118,-61.463,-178.441,7.328,148.924
C09925=1136.470,176.870,-61.441,-178.444,7.325,148.925
C09926=1136.476,176.621,-61.418,-178.447,7.323,148.925
C09927=1136.480,176.372,-61.396,-178.450,7.321,148.925
C09928=1136.485,176.123,-61.372,-178.452,7.318,148.925
C09929=1136.489,175.874,-61.349,-178.455,7.316,148.926
C09930=1136.494,175.625,-61.327,-178.458,7.314,148.926
C09931=1136.498,175.377,-61.304,-178.461,7.311,148.926
C09932=1136.503,175.128,-61.281,-178.464,7.310,148.927
C09933=1136.508,174.879,-61.259,-178.467,7.307,148.927
C09934=1136.513,174.630,-61.236,-178.469,7.305,148.927
C09935=1136.517,174.381,-61.214,-178.472,7.302,148.927
C09936=1136.522,174.132,-61.191,-178.475,7.300,148.928
C09937=1136.526,173.884,-61.168,-178.478,7.298,148.928
C09938=1136.531,173.634,-61.146,-178.481,7.296,148.928
C09939=1136.535,173.385,-61.123,-178.484,7.293,148.928
C09940=1136.541,173.136,-61.101,-178.486,7.292,148.929
C09941=1136.545,172.887,-61.078,-178.490,7.289,148.929
C09942=1136.550,172.638,-61.055,-178.492,7.287,148.929
C09943=1136.554,172.390,-61.033,-178.495,7.284,148.930
C09944=1136.559,172.140,-61.010,-178.497,7.282,148.930
C09945=1136.563,171.891,-60.987,-178.501,7.280,148.930
C09946=1136.568,171.643,-60.966,-178.503,7.278,148.931
C09947=1136.573,171.393,-60.943,-178.506,7.275,148.931
C09948=1136.577,171.144,-60.920,-178.509,7.273,148.931
C09949=1136.583,170.895,-60.898,-178.512,7.271,148.931
C09950=1136.587,170.647,-60.875,-178.514,7.269,148.932
C09951=1136.591,170.398,-60.854,-178.518,7.266,148.932
C09952=1136.596,170.148,-60.831,-178.520,7.265,148.932
C09953=1136.600,169.900,-60.808,-178.523,7.262,148.932
C09954=1136.605,169.651,-60.786,-178.526,7.260,148.933
C09955=1136.610,169.401,-60.764,-178.529,7.258,148.933
C09956=1136.615,169.153,-60.741,-178.531,7.255,148.933
C09957=1136.619,168.904,-60.719,-178.535,7.253,148.934
C09958=1136.624,168.654,-60.697,-178.537,7.251,148.934
C09959=1136.629,168.406,-60.674,-178.540,7.248,148.934
C09960=1136.633,168.157,-60.652,-178.543,7.247,148.934
C09961=1136.638,167.908,-60.631,-178.546,7.245,148.935
C09962=1136.643,167.659,-60.608,-178.549,7.242,148.935
C09963=1136.647,167.411,-60.586,-178.551,7.240,148.935
C09964=1136.652,167.161,-60.563,-178.555,7.238,148.936
C09965=1136.657,166.912,-60.541,-178.557,7.236,148.936
C09966=1136.662,166.663,-60.519,-178.560,7.233,148.936
C09967=1136.666,166.414,-60.497,-178.563,7.231,148.937
C09968=1136.670,166.166,-60.475,-178.566,7.229,148.937
C09969=1136.675,165.916,-60.452,-178.568,7.227,148.937
C09970=1136.680,165.667,-60.430,-178.572,7.224,148.937
C09971=1136.684,165.418,-60.408,-178.574,7.222,148.938
C09972=1136.689,165.169,-60.387,-178.577,7.221,148.938
C09973=1136.694,164.920,-60.365,-178.580,7.218,148.938
C09974=1136.699,164.671,-60.343,-178.583,7.216,148.939
C09975=1136.704,164.422,-60.320,-178.585,7.213,148.939
C09976=1136.708,164.173,-60.299,-178.588,7.212,148.939
C09977=1136.712,163.924,-60.276,-178.591,7.209,148.940
C09978=1136.717,163.676,-60.254,-178.594,7.207,148.940
C09979=1136.721,163.426,-60.232,-178.596,7.205,148.940
C09980=1136.726,163.178,-60.210,-178.600,7.203,148.940
C09981=1136.731,162.929,-60.188,-178.602,7.201,148.941
C09982=1136.735,162.680,-60.167,-178.605,7.198,148.941
C09983=1136.741,162.431,-60.144,-178.608,7.197,148.941
C09984=1136.745,162.182,-60.122,-178.611,7.194,148.942
C09985=1136.750,161.933,-60.101,-178.613,7.192,148.942
C09986=1136.754,161.684,-60.079,-178.616,7.190,148.942
C09987=1136.759,161.435,-60.057,-178.619,7.188,148.943
C09988=1136.764,161.185,-60.036,-178.622,7.186,148.943
C09989=1136.769,160.936,-60.014,-178.625,7.183,148.943
C09990=1136.774,160.688,-59.992,-178.628,7.181,148.944
C09991=1136.778,160.438,-59.970,-178.630,7.180,148.944
C09992=1136.783,160.190,-59.949,-178.633,7.177,148.944
C09993=1136.787,159.940,-59.926,-178.636,7.175,148.944
C09994=1136.792,159.692,-59.905,-178.639,7.173,148.945
C09995=1136.796,159.442,-59.883,-178.642,7.171,148.945
C09996=1136.801,159.193,-59.862,-178.644,7.169,148.945
//INST
///DATE 2021/06/25 14:32
///ATTR SC,RW,RJ
////FRAME ROBOT
///GROUP1 RB1
NOP
MOVL C00000 V=800.0 PL=0
MOVL C00001 V=800.0 PL=0
MOVL C00002 V=800.0 PL=0
MOVL C00003 V=800.0 PL=0
MOVL C00004 V=800.0 PL=0
MOVL C00005 V=800.0 PL=0
MOVL C00006 V=800.0 PL=0
MOVL C00007 V=800.0 PL=0
MOVL C00008 V=800.0 PL=0
MOVL C00009 V=800.0 PL=0
MOVL C00010 V=800.0 PL=0
MOVL C00011 V=800.0 PL=0
MOVL C00012 V=800.0 PL=0
MOVL C00013 V=800.0 PL=0
MOVL C00014 V=800.0 PL=0
MOVL C00015 V=800.0 PL=0
MOVL C00016 V=800.0 PL=0
MOVL C00017 V=800.0 PL=0
MOVL C00018 V=800.0 PL=0
MOVL C00019 V=800.0 PL=0
MOVL C00020 V=800.0 PL=0
MOVL C00021 V=800.0 PL=0
MOVL C00022 V=800.0 PL=0
MOVL C00023 V=800.0 PL=0
MOVL C00024 V=800.0 PL=0
MOVL C00025 V=800.0 PL=0
MOVL C00026 V=800.0 PL=0
MOVL C00027 V=800.0 PL=0
MOVL C00028 V=800.0 PL=0
MOVL C00029 V=800.0 PL=0
MOVL C00030 V=800.0 PL=0
MOVL C00031 V=800.0 PL=0
MOVL C00032 V=800.0 PL=0
MOVL C00033 V=800.0 PL=0
MOVL C00034 V=800.0 PL=0
MOVL C00035 V=800.0 PL=0
MOVL C00036 V=800.0 PL=0
MOVL C00037 V=800.0 PL=0
MOVL C00038 V=800.0 PL=0
MOVL C00039 V=800.0 PL=0
MOVL C00040 V=800.0 PL=0
MOVL C00041 V=800.0 PL=0
MOVL C00042 V=800.0 PL=0
MOVL C00043 V=800.0 PL=0
MOVL C00044 V=800.0 PL=0
MOVL C00045 V=800.0 PL=0
MOVL C00046 V=800.0 PL=0
MOVL C00047 V=800.0 PL=0
MOVL C00048 V=800.0 PL=0
MOVL C00049 V=800.0 PL=0
MOVL C00050 V=800.0 PL=0
MOVL C00051 V=800.0 PL=0
MOVL C00052 V=800.0 PL=0
MOVL C00053 V=800.0 PL=0
MOVL C00054 V=800.0 PL=0
MOVL C00055 V=800.0 PL=0
MOVL C00056 V=800.0 PL=0
MOVL C00057 V=800.0 PL=0
MOVL C00058 V=800.0 PL=0
MOVL C00059 V=800.0 PL=0
MOVL C00060 V=800.0 PL=0
MOVL C00061 V=800.0 PL=0
MOVL C00062 V=800.0 PL=0
MOVL C00063 V=800.0 PL=0
MOVL C00064 V=800.0 PL=0
MOVL C00065 V=800.0 PL=0
MOVL C00066 V=800.0 PL=0
MOVL C00067 V=800.0 PL=0
MOVL C00068 V=800.0 PL=0
MOVL C00069 V=800.0 PL=0
MOVL C00070 V=800.0 PL=0
MOVL C00071 V=800.0 PL=0
MOVL C00072 V=800.0 PL=0
MOVL C00073 V=800.0 PL=0
MOVL C00074 V=800.0 PL=0
MOVL C00075 V=800.0 PL=0
MOVL C00076 V=800.0 PL=0
MOVL C00077 V=800.0 PL=0
MOVL C00078 V=800.0 PL=0
MOVL C00079 V=800.0 PL=0
MOVL C00080 V=800.0 PL=0
MOVL C00081 V=800.0 PL=0
MOVL C00082 V=800.0 PL=0
MOVL C00083 V=800.0 PL=0
MOVL C00084 V=800.0 PL=0
MOVL C00085 V=800.0 PL=0
MOVL C00086 V=800.0 PL=0
MOVL C00087 V=800.0 PL=0
MOVL C00088 V=800.0 PL=0
MOVL C00089 V=800.0 PL=0
MOVL C00090 V=800.0 PL=0
MOVL C00091 V=800.0 PL=0
MOVL C00092 V=800.0 PL=0
MOVL C00093 V=800.0 PL=0
MOVL C00094 V=800.0 PL=0
MOVL C00095 V=800.0 PL=0
MOVL C00096 V=800.0 PL=0
MOVL C00097 V=800.0 PL=0
MOVL C00098 V=800.0 PL=0
MOVL C00099 V=800.0 PL=0
MOVL C00100 V=800.0 PL=0
MOVL C00101 V=800.0 PL=0
MOVL C00102 V=800.0 PL=0
MOVL C00103 V=800.0 PL=0
MOVL C00104 V=800.0 PL=0
MOVL C00105 V=800.0 PL=0
MOVL C00106 V=800.0 PL=0
MOVL C00107 V=800.0 PL=0
MOVL C00108 V=800.0 PL=0
MOVL C00109 V=800.0 PL=0
MOVL C00110 V=800.0 PL=0
MOVL C00111 V=800.0 PL=0
MOVL C00112 V=800.0 PL=0
MOVL C00113 V=800.0 PL=0
MOVL C00114 V=800.0 PL=0
MOVL C00115 V=800.0 PL=0
MOVL C00116 V=800.0 PL=0
MOVL C00117 V=800.0 PL=0
MOVL C00118 V=800.0 PL=0
MOVL C00119 V=800.0 PL=0
MOVL C00120 V=800.0 PL=0
MOVL C00121 V=800.0 PL=0
MOVL C00122 V=800.0 PL=0
MOVL C00123 V=800.0 PL=0
MOVL C00124 V=800.0 PL=0
MOVL C00125 V=800.0 PL=0
MOVL C00126 V=800.0 PL=0
MOVL C00127 V=800.0 PL=0
MOVL C00128 V=800.0 PL=0
MOVL C00129 V=800.0 PL=0
MOVL C00130 V=800.0 PL=0
MOVL C00131 V=800.0 PL=0
MOVL C00132 V=800.0 PL=0
MOVL C00133 V=800.0 PL=0
MOVL C00134 V=800.0 PL=0
MOVL C00135 V=800.0 PL=0
MOVL C00136 V=800.0 PL=0
MOVL C00137 V=800.0 PL=0
MOVL C00138 V=800.0 PL=0
MOVL C00139 V=800.0 PL=0
MOVL C00140 V=800.0 PL=0
MOVL C00141 V=800.0 PL=0
MOVL C00142 V=800.0 PL=0
MOVL C00143 V=800.0 PL=0
MOVL C00144 V=800.0 PL=0
MOVL C00145 V=800.0 PL=0
MOVL C00146 V=800.0 PL=0
MOVL C00147 V=800.0 PL=0
MOVL C00148 V=800.0 PL=0
MOVL C00149 V=800.0 PL=0
MOVL C00150 V=800.0 PL=0
MOVL C00151 V=800.0 PL=0
MOVL C00152 V=800.0 PL=0
MOVL C00153 V=800.0 PL=0
MOVL C00154 V=800.0 PL=0
MOVL C00155 V=800.0 PL=0
MOVL C00156 V=800.0 PL=0
MOVL C00157 V=800.0 PL=0
MOVL C00158 V=800.0 PL=0
MOVL C00159 V=800.0 PL=0
MOVL C00160 V=800.0 PL=0
MOVL C00161 V=800.0 PL=0
MOVL C00162 V=800.0 PL=0
MOVL C00163 V=800.0 PL=0
MOVL C00164 V=800.0 PL=0
MOVL C00165 V=800.0 PL=0
MOVL C00166 V=800.0 PL=0
MOVL C00167 V=800.0 PL=0
MOVL C00168 V=800.0 PL=0
MOVL C00169 V=800.0 PL=0
MOVL C00170 V=800.0 PL=0
MOVL C00171 V=800.0 PL=0
MOVL C00172 V=800.0 PL=0
MOVL C00173 V=800.0 PL=0
MOVL C00174 V=800.0 PL=0
MOVL C00175 V=800.0 PL=0
MOVL C00176 V=800.0 PL=0
MOVL C00177 V=800.0 PL=0
MOVL C00178 V=800.0 PL=0
MOVL C00179 V=800.0 PL=0
MOVL C00180 V=800.0 PL=0
MOVL C00181 V=800.0 PL=0
MOVL C00182 V=800.0 PL=0
MOVL C00183 V=800.0 PL=0
MOVL C00184 V=800.0 PL=0
MOVL C00185 V=800.0 PL=0
MOVL C00186 V=800.0 PL=0
MOVL C00187 V=800.0 PL=0
MOVL C00188 V=800.0 PL=0
MOVL C00189 V=800.0 PL=0
MOVL C00190 V=800.0 PL=0
MOVL C00191 V=800.0 PL=0
MOVL C00192 V=800.0 PL=0
MOVL C00193 V=800.0 PL=0
MOVL C00194 V=800.0 PL=0
MOVL C00195 V=800.0 PL=0
MOVL C00196 V=800.0 PL=0
MOVL C00197 V=800.0 PL=0
MOVL C00198 V=800.0 PL=0
MOVL C00199 V=800.0 PL=0
MOVL C00200 V=800.0 PL=0
MOVL C00201 V=800.0 PL=0
MOVL C00202 V=800.0 PL=0
MOVL C00203 V=800.0 PL=0
MOVL C00204 V=800.0 PL=0
MOVL C00205 V=800.0 PL=0
MOVL C00206 V=800.0 PL=0
MOVL C00207 V=800.0 PL=0
MOVL C00208 V=800.0 PL=0
MOVL C00209 V=800.0 PL=0
MOVL C00210 V=800.0 PL=0
MOVL C00211 V=800.0 PL=0
MOVL C00212 V=800.0 PL=0
MOVL C00213 V=800.0 PL=0
MOVL C00214 V=800.0 PL=0
MOVL C00215 V=800.0 PL=0
MOVL C00216 V=800.0 PL=0
MOVL C00217 V=800.0 PL=0
MOVL C00218 V=800.0 PL=0
MOVL C00219 V=800.0 PL=0
MOVL C00220 V=800.0 PL=0
MOVL C00221 V=800.0 PL=0
MOVL C00222 V=800.0 PL=0
MOVL C00223 V=800.0 PL=0
MOVL C00224 V=800.0 PL=0
MOVL C00225 V=800.0 PL=0
MOVL C00226 V=800.0 PL=0
MOVL C00227 V=800.0 PL=0
MOVL C00228 V=800.0 PL=0
MOVL C00229 V=800.0 PL=0
MOVL C00230 V=800.0 PL=0
MOVL C00231 V=800.0 PL=0
MOVL C00232 V=800.0 PL=0
MOVL C00233 V=800.0 PL=0
MOVL C00234 V=800.0 PL=0
MOVL C00235 V=800.0 PL=0
MOVL C00236 V=800.0 PL=0
MOVL C00237 V=800.0 PL=0
MOVL C00238 V=800.0 PL=0
MOVL C00239 V=800.0 PL=0
MOVL C00240 V=800.0 PL=0
MOVL C00241 V=800.0 PL=0
MOVL C00242 V=800.0 PL=0
MOVL C00243 V=800.0 PL=0
MOVL C00244 V=800.0 PL=0
MOVL C00245 V=800.0 PL=0
MOVL C00246 V=800.0 PL=0
MOVL C00247 V=800.0 PL=0
MOVL C00248 V=800.0 PL=0
MOVL C00249 V=800.0 PL=0
MOVL C00250 V=800.0 PL=0
MOVL C00251 V=800.0 PL=0
MOVL C00252 V=800.0 PL=0
MOVL C00253 V=800.0 PL=0
MOVL C00254 V=800.0 PL=0
MOVL C00255 V=800.0 PL=0
MOVL C00256 V=800.0 PL=0
MOVL C00257 V=800.0 PL=0
MOVL C00258 V=800.0 PL=0
MOVL C00259 V=800.0 PL=0
MOVL C00260 V=800.0 PL=0
MOVL C00261 V=800.0 PL=0
MOVL C00262 V=800.0 PL=0
MOVL C00263 V=800.0 PL=0
MOVL C00264 V=800.0 PL=0
MOVL C00265 V=800.0 PL=0
MOVL C00266 V=800.0 PL=0
MOVL C00267 V=800.0 PL=0
MOVL C00268 V=800.0 PL=0
MOVL C00269 V=800.0 PL=0
MOVL C00270 V=800.0 PL=0
MOVL C00271 V=800.0 PL=0
MOVL C00272 V=800.0 PL=0
MOVL C00273 V=800.0 PL=0
MOVL C00274 V=800.0 PL=0
MOVL C00275 V=800.0 PL=0
MOVL C00276 V=800.0 PL=0
MOVL C00277 V=800.0 PL=0
MOVL C00278 V=800.0 PL=0
MOVL C00279 V=800.0 PL=0
MOVL C00280 V=800.0 PL=0
MOVL C00281 V=800.0 PL=0
MOVL C00282 V=800.0 PL=0
MOVL C00283 V=800.0 PL=0
MOVL C00284 V=800.0 PL=0
MOVL C00285 V=800.0 PL=0
MOVL C00286 V=800.0 PL=0
MOVL C00287 V=800.0 PL=0
MOVL C00288 V=800.0 PL=0
MOVL C00289 V=800.0 PL=0
MOVL C00290 V=800.0 PL=0
MOVL C00291 V=800.0 PL=0
MOVL C00292 V=800.0 PL=0
MOVL C00293 V=800.0 PL=0
MOVL C00294 V=800.0 PL=0
MOVL C00295 V=800.0 PL=0
MOVL C00296 V=800.0 PL=0
MOVL C00297 V=800.0 PL=0
MOVL C00298 V=800.0 PL=0
MOVL C00299 V=800.0 PL=0
MOVL C00300 V=800.0 PL=0
MOVL C00301 V=800.0 PL=0
MOVL C00302 V=800.0 PL=0
MOVL C00303 V=800.0 PL=0
MOVL C00304 V=800.0 PL=0
MOVL C00305 V=800.0 PL=0
MOVL C00306 V=800.0 PL=0
MOVL C00307 V=800.0 PL=0
MOVL C00308 V=800.0 PL=0
MOVL C00309 V=800.0 PL=0
MOVL C00310 V=800.0 PL=0
MOVL C00311 V=800.0 PL=0
MOVL C00312 V=800.0 PL=0
MOVL C00313 V=800.0 PL=0
MOVL C00314 V=800.0 PL=0
MOVL C00315 V=800.0 PL=0
MOVL C00316 V=800.0 PL=0
MOVL C00317 V=800.0 PL=0
MOVL C00318 V=800.0 PL=0
MOVL C00319 V=800.0 PL=0
MOVL C00320 V=800.0 PL=0
MOVL C00321 V=800.0 PL=0
MOVL C00322 V=800.0 PL=0
MOVL C00323 V=800.0 PL=0
MOVL C00324 V=800.0 PL=0
MOVL C00325 V=800.0 PL=0
MOVL C00326 V=800.0 PL=0
MOVL C00327 V=800.0 PL=0
MOVL C00328 V=800.0 PL=0
MOVL C00329 V=800.0 PL=0
MOVL C00330 V=800.0 PL=0
MOVL C00331 V=800.0 PL=0
MOVL C00332 V=800.0 PL=0
MOVL C00333 V=800.0 PL=0
MOVL C00334 V=800.0 PL=0
MOVL C00335 V=800.0 PL=0
MOVL C00336 V=800.0 PL=0
MOVL C00337 V=800.0 PL=0
MOVL C00338 V=800.0 PL=0
MOVL C00339 V=800.0 PL=0
MOVL C00340 V=800.0 PL=0
MOVL C00341 V=800.0 PL=0
MOVL C00342 V=800.0 PL=0
MOVL C00343 V=800.0 PL=0
MOVL C00344 V=800.0 PL=0
MOVL C00345 V=800.0 PL=0
MOVL C00346 V=800.0 PL=0
MOVL C00347 V=800.0 PL=0
MOVL C00348 V=800.0 PL=0
MOVL C00349 V=800.0 PL=0
MOVL C00350 V=800.0 PL=0
MOVL C00351 V=800.0 PL=0
MOVL C00352 V=800.0 PL=0
MOVL C00353 V=800.0 PL=0
MOVL C00354 V=800.0 PL=0
MOVL C00355 V=800.0 PL=0
MOVL C00356 V=800.0 PL=0
MOVL C00357 V=800.0 PL=0
MOVL C00358 V=800.0 PL=0
MOVL C00359 V=800.0 PL=0
MOVL C00360 V=800.0 PL=0
MOVL C00361 V=800.0 PL=0
MOVL C00362 V=800.0 PL=0
MOVL C00363 V=800.0 PL=0
MOVL C00364 V=800.0 PL=0
MOVL C00365 V=800.0 PL=0
MOVL C00366 V=800.0 PL=0
MOVL C00367 V=800.0 PL=0
MOVL C00368 V=800.0 PL=0
MOVL C00369 V=800.0 PL=0
MOVL C00370 V=800.0 PL=0
MOVL C00371 V=800.0 PL=0
MOVL C00372 V=800.0 PL=0
MOVL C00373 V=800.0 PL=0
MOVL C00374 V=800.0 PL=0
MOVL C00375 V=800.0 PL=0
MOVL C00376 V=800.0 PL=0
MOVL C00377 V=800.0 PL=0
MOVL C00378 V=800.0 PL=0
MOVL C00379 V=800.0 PL=0
MOVL C00380 V=800.0 PL=0
MOVL C00381 V=800.0 PL=0
MOVL C00382 V=800.0 PL=0
MOVL C00383 V=800.0 PL=0
MOVL C00384 V=800.0 PL=0
MOVL C00385 V=800.0 PL=0
MOVL C00386 V=800.0 PL=0
MOVL C00387 V=800.0 PL=0
MOVL C00388 V=800.0 PL=0
MOVL C00389 V=800.0 PL=0
MOVL C00390 V=800.0 PL=0
MOVL C00391 V=800.0 PL=0
MOVL C00392 V=800.0 PL=0
MOVL C00393 V=800.0 PL=0
MOVL C00394 V=800.0 PL=0
MOVL C00395 V=800.0 PL=0
MOVL C00396 V=800.0 PL=0
MOVL C00397 V=800.0 PL=0
MOVL C00398 V=800.0 PL=0
MOVL C00399 V=800.0 PL=0
MOVL C00400 V=800.0 PL=0
MOVL C00401 V=800.0 PL=0
MOVL C00402 V=800.0 PL=0
MOVL C00403 V=800.0 PL=0
MOVL C00404 V=800.0 PL=0
MOVL C00405 V=800.0 PL=0
MOVL C00406 V=800.0 PL=0
MOVL C00407 V=800.0 PL=0
MOVL C00408 V=800.0 PL=0
MOVL C00409 V=800.0 PL=0
MOVL C00410 V=800.0 PL=0
MOVL C00411 V=800.0 PL=0
MOVL C00412 V=800.0 PL=0
MOVL C00413 V=800.0 PL=0
MOVL C00414 V=800.0 PL=0
MOVL C00415 V=800.0 PL=0
MOVL C00416 V=800.0 PL=0
MOVL C00417 V=800.0 PL=0
MOVL C00418 V=800.0 PL=0
MOVL C00419 V=800.0 PL=0
MOVL C00420 V=800.0 PL=0
MOVL C00421 V=800.0 PL=0
MOVL C00422 V=800.0 PL=0
MOVL C00423 V=800.0 PL=0
MOVL C00424 V=800.0 PL=0
MOVL C00425 V=800.0 PL=0
MOVL C00426 V=800.0 PL=0
MOVL C00427 V=800.0 PL=0
MOVL C00428 V=800.0 PL=0
MOVL C00429 V=800.0 PL=0
MOVL C00430 V=800.0 PL=0
MOVL C00431 V=800.0 PL=0
MOVL C00432 V=800.0 PL=0
MOVL C00433 V=800.0 PL=0
MOVL C00434 V=800.0 PL=0
MOVL C00435 V=800.0 PL=0
MOVL C00436 V=800.0 PL=0
MOVL C00437 V=800.0 PL=0
MOVL C00438 V=800.0 PL=0
MOVL C00439 V=800.0 PL=0
MOVL C00440 V=800.0 PL=0
MOVL C00441 V=800.0 PL=0
MOVL C00442 V=800.0 PL=0
MOVL C00443 V=800.0 PL=0
MOVL C00444 V=800.0 PL=0
MOVL C00445 V=800.0 PL=0
MOVL C00446 V=800.0 PL=0
MOVL C00447 V=800.0 PL=0
MOVL C00448 V=800.0 PL=0
MOVL C00449 V=800.0 PL=0
MOVL C00450 V=800.0 PL=0
MOVL C00451 V=800.0 PL=0
MOVL C00452 V=800.0 PL=0
MOVL C00453 V=800.0 PL=0
MOVL C00454 V=800.0 PL=0
MOVL C00455 V=800.0 PL=0
MOVL C00456 V=800.0 PL=0
MOVL C00457 V=800.0 PL=0
MOVL C00458 V=800.0 PL=0
MOVL C00459 V=800.0 PL=0
MOVL C00460 V=800.0 PL=0
MOVL C00461 V=800.0 PL=0
MOVL C00462 V=800.0 PL=0
MOVL C00463 V=800.0 PL=0
MOVL C00464 V=800.0 PL=0
MOVL C00465 V=800.0 PL=0
MOVL C00466 V=800.0 PL=0
MOVL C00467 V=800.0 PL=0
MOVL C00468 V=800.0 PL=0
MOVL C00469 V=800.0 PL=0
MOVL C00470 V=800.0 PL=0
MOVL C00471 V=800.0 PL=0
MOVL C00472 V=800.0 PL=0
MOVL C00473 V=800.0 PL=0
MOVL C00474 V=800.0 PL=0
MOVL C00475 V=800.0 PL=0
MOVL C00476 V=800.0 PL=0
MOVL C00477 V=800.0 PL=0
MOVL C00478 V=800.0 PL=0
MOVL C00479 V=800.0 PL=0
MOVL C00480 V=800.0 PL=0
MOVL C00481 V=800.0 PL=0
MOVL C00482 V=800.0 PL=0
MOVL C00483 V=800.0 PL=0
MOVL C00484 V=800.0 PL=0
MOVL C00485 V=800.0 PL=0
MOVL C00486 V=800.0 PL=0
MOVL C00487 V=800.0 PL=0
MOVL C00488 V=800.0 PL=0
MOVL C00489 V=800.0 PL=0
MOVL C00490 V=800.0 PL=0
MOVL C00491 V=800.0 PL=0
MOVL C00492 V=800.0 PL=0
MOVL C00493 V=800.0 PL=0
MOVL C00494 V=800.0 PL=0
MOVL C00495 V=800.0 PL=0
MOVL C00496 V=800.0 PL=0
MOVL C00497 V=800.0 PL=0
MOVL C00498 V=800.0 PL=0
MOVL C00499 V=800.0 PL=0
MOVL C00500 V=800.0 PL=0
MOVL C00501 V=800.0 PL=0
MOVL C00502 V=800.0 PL=0
MOVL C00503 V=800.0 PL=0
MOVL C00504 V=800.0 PL=0
MOVL C00505 V=800.0 PL=0
MOVL C00506 V=800.0 PL=0
MOVL C00507 V=800.0 PL=0
MOVL C00508 V=800.0 PL=0
MOVL C00509 V=800.0 PL=0
MOVL C00510 V=800.0 PL=0
MOVL C00511 V=800.0 PL=0
MOVL C00512 V=800.0 PL=0
MOVL C00513 V=800.0 PL=0
MOVL C00514 V=800.0 PL=0
MOVL C00515 V=800.0 PL=0
MOVL C00516 V=800.0 PL=0
MOVL C00517 V=800.0 PL=0
MOVL C00518 V=800.0 PL=0
MOVL C00519 V=800.0 PL=0
MOVL C00520 V=800.0 PL=0
MOVL C00521 V=800.0 PL=0
MOVL C00522 V=800.0 PL=0
MOVL C00523 V=800.0 PL=0
MOVL C00524 V=800.0 PL=0
MOVL C00525 V=800.0 PL=0
MOVL C00526 V=800.0 PL=0
MOVL C00527 V=800.0 PL=0
MOVL C00528 V=800.0 PL=0
MOVL C00529 V=800.0 PL=0
MOVL C00530 V=800.0 PL=0
MOVL C00531 V=800.0 PL=0
MOVL C00532 V=800.0 PL=0
MOVL C00533 V=800.0 PL=0
MOVL C00534 V=800.0 PL=0
MOVL C00535 V=800.0 PL=0
MOVL C00536 V=800.0 PL=0
MOVL C00537 V=800.0 PL=0
MOVL C00538 V=800.0 PL=0
MOVL C00539 V=800.0 PL=0
MOVL C00540 V=800.0 PL=0
MOVL C00541 V=800.0 PL=0
MOVL C00542 V=800.0 PL=0
MOVL C00543 V=800.0 PL=0
MOVL C00544 V=800.0 PL=0
MOVL C00545 V=800.0 PL=0
MOVL C00546 V=800.0 PL=0
MOVL C00547 V=800.0 PL=0
MOVL C00548 V=800.0 PL=0
MOVL C00549 V=800.0 PL=0
MOVL C00550 V=800.0 PL=0
MOVL C00551 V=800.0 PL=0
MOVL C00552 V=800.0 PL=0
MOVL C00553 V=800.0 PL=0
MOVL C00554 V=800.0 PL=0
MOVL C00555 V=800.0 PL=0
MOVL C00556 V=800.0 PL=0
MOVL C00557 V=800.0 PL=0
MOVL C00558 V=800.0 PL=0
MOVL C00559 V=800.0 PL=0
MOVL C00560 V=800.0 PL=0
MOVL C00561 V=800.0 PL=0
MOVL C00562 V=800.0 PL=0
MOVL C00563 V=800.0 PL=0
MOVL C00564 V=800.0 PL=0
MOVL C00565 V=800.0 PL=0
MOVL C00566 V=800.0 PL=0
MOVL C00567 V=800.0 PL=0
MOVL C00568 V=800.0 PL=0
MOVL C00569 V=800.0 PL=0
MOVL C00570 V=800.0 PL=0
MOVL C00571 V=800.0 PL=0
MOVL C00572 V=800.0 PL=0
MOVL C00573 V=800.0 PL=0
MOVL C00574 V=800.0 PL=0
MOVL C00575 V=800.0 PL=0
MOVL C00576 V=800.0 PL=0
MOVL C00577 V=800.0 PL=0
MOVL C00578 V=800.0 PL=0
MOVL C00579 V=800.0 PL=0
MOVL C00580 V=800.0 PL=0
MOVL C00581 V=800.0 PL=0
MOVL C00582 V=800.0 PL=0
MOVL C00583 V=800.0 PL=0
MOVL C00584 V=800.0 PL=0
MOVL C00585 V=800.0 PL=0
MOVL C00586 V=800.0 PL=0
MOVL C00587 V=800.0 PL=0
MOVL C00588 V=800.0 PL=0
MOVL C00589 V=800.0 PL=0
MOVL C00590 V=800.0 PL=0
MOVL C00591 V=800.0 PL=0
MOVL C00592 V=800.0 PL=0
MOVL C00593 V=800.0 PL=0
MOVL C00594 V=800.0 PL=0
MOVL C00595 V=800.0 PL=0
MOVL C00596 V=800.0 PL=0
MOVL C00597 V=800.0 PL=0
MOVL C00598 V=800.0 PL=0
MOVL C00599 V=800.0 PL=0
MOVL C00600 V=800.0 PL=0
MOVL C00601 V=800.0 PL=0
MOVL C00602 V=800.0 PL=0
MOVL C00603 V=800.0 PL=0
MOVL C00604 V=800.0 PL=0
MOVL C00605 V=800.0 PL=0
MOVL C00606 V=800.0 PL=0
MOVL C00607 V=800.0 PL=0
MOVL C00608 V=800.0 PL=0
MOVL C00609 V=800.0 PL=0
MOVL C00610 V=800.0 PL=0
MOVL C00611 V=800.0 PL=0
MOVL C00612 V=800.0 PL=0
MOVL C00613 V=800.0 PL=0
MOVL C00614 V=800.0 PL=0
MOVL C00615 V=800.0 PL=0
MOVL C00616 V=800.0 PL=0
MOVL C00617 V=800.0 PL=0
MOVL C00618 V=800.0 PL=0
MOVL C00619 V=800.0 PL=0
MOVL C00620 V=800.0 PL=0
MOVL C00621 V=800.0 PL=0
MOVL C00622 V=800.0 PL=0
MOVL C00623 V=800.0 PL=0
MOVL C00624 V=800.0 PL=0
MOVL C00625 V=800.0 PL=0
MOVL C00626 V=800.0 PL=0
MOVL C00627 V=800.0 PL=0
MOVL C00628 V=800.0 PL=0
MOVL C00629 V=800.0 PL=0
MOVL C00630 V=800.0 PL=0
MOVL C00631 V=800.0 PL=0
MOVL C00632 V=800.0 PL=0
MOVL C00633 V=800.0 PL=0
MOVL C00634 V=800.0 PL=0
MOVL C00635 V=800.0 PL=0
MOVL C00636 V=800.0 PL=0
MOVL C00637 V=800.0 PL=0
MOVL C00638 V=800.0 PL=0
MOVL C00639 V=800.0 PL=0
MOVL C00640 V=800.0 PL=0
MOVL C00641 V=800.0 PL=0
MOVL C00642 V=800.0 PL=0
MOVL C00643 V=800.0 PL=0
MOVL C00644 V=800.0 PL=0
MOVL C00645 V=800.0 PL=0
MOVL C00646 V=800.0 PL=0
MOVL C00647 V=800.0 PL=0
MOVL C00648 V=800.0 PL=0
MOVL C00649 V=800.0 PL=0
MOVL C00650 V=800.0 PL=0
MOVL C00651 V=800.0 PL=0
MOVL C00652 V=800.0 PL=0
MOVL C00653 V=800.0 PL=0
MOVL C00654 V=800.0 PL=0
MOVL C00655 V=800.0 PL=0
MOVL C00656 V=800.0 PL=0
MOVL C00657 V=800.0 PL=0
MOVL C00658 V=800.0 PL=0
MOVL C00659 V=800.0 PL=0
MOVL C00660 V=800.0 PL=0
MOVL C00661 V=800.0 PL=0
MOVL C00662 V=800.0 PL=0
MOVL C00663 V=800.0 PL=0
MOVL C00664 V=800.0 PL=0
MOVL C00665 V=800.0 PL=0
MOVL C00666 V=800.0 PL=0
MOVL C00667 V=800.0 PL=0
MOVL C00668 V=800.0 PL=0
MOVL C00669 V=800.0 PL=0
MOVL C00670 V=800.0 PL=0
MOVL C00671 V=800.0 PL=0
MOVL C00672 V=800.0 PL=0
MOVL C00673 V=800.0 PL=0
MOVL C00674 V=800.0 PL=0
MOVL C00675 V=800.0 PL=0
MOVL C00676 V=800.0 PL=0
MOVL C00677 V=800.0 PL=0
MOVL C00678 V=800.0 PL=0
MOVL C00679 V=800.0 PL=0
MOVL C00680 V=800.0 PL=0
MOVL C00681 V=800.0 PL=0
MOVL C00682 V=800.0 PL=0
MOVL C00683 V=800.0 PL=0
MOVL C00684 V=800.0 PL=0
MOVL C00685 V=800.0 PL=0
MOVL C00686 V=800.0 PL=0
MOVL C00687 V=800.0 PL=0
MOVL C00688 V=800.0 PL=0
MOVL C00689 V=800.0 PL=0
MOVL C00690 V=800.0 PL=0
MOVL C00691 V=800.0 PL=0
MOVL C00692 V=800.0 PL=0
MOVL C00693 V=800.0 PL=0
MOVL C00694 V=800.0 PL=0
MOVL C00695 V=800.0 PL=0
MOVL C00696 V=800.0 PL=0
MOVL C00697 V=800.0 PL=0
MOVL C00698 V=800.0 PL=0
MOVL C00699 V=800.0 PL=0
MOVL C00700 V=800.0 PL=0
MOVL C00701 V=800.0 PL=0
MOVL C00702 V=800.0 PL=0
MOVL C00703 V=800.0 PL=0
MOVL C00704 V=800.0 PL=0
MOVL C00705 V=800.0 PL=0
MOVL C00706 V=800.0 PL=0
MOVL C00707 V=800.0 PL=0
MOVL C00708 V=800.0 PL=0
MOVL C00709 V=800.0 PL=0
MOVL C00710 V=800.0 PL=0
MOVL C00711 V=800.0 PL=0
MOVL C00712 V=800.0 PL=0
MOVL C00713 V=800.0 PL=0
MOVL C00714 V=800.0 PL=0
MOVL C00715 V=800.0 PL=0
MOVL C00716 V=800.0 PL=0
MOVL C00717 V=800.0 PL=0
MOVL C00718 V=800.0 PL=0
MOVL C00719 V=800.0 PL=0
MOVL C00720 V=800.0 PL=0
MOVL C00721 V=800.0 PL=0
MOVL C00722 V=800.0 PL=0
MOVL C00723 V=800.0 PL=0
MOVL C00724 V=800.0 PL=0
MOVL C00725 V=800.0 PL=0
MOVL C00726 V=800.0 PL=0
MOVL C00727 V=800.0 PL=0
MOVL C00728 V=800.0 PL=0
MOVL C00729 V=800.0 PL=0
MOVL C00730 V=800.0 PL=0
MOVL C00731 V=800.0 PL=0
MOVL C00732 V=800.0 PL=0
MOVL C00733 V=800.0 PL=0
MOVL C00734 V=800.0 PL=0
MOVL C00735 V=800.0 PL=0
MOVL C00736 V=800.0 PL=0
MOVL C00737 V=800.0 PL=0
MOVL C00738 V=800.0 PL=0
MOVL C00739 V=800.0 PL=0
MOVL C00740 V=800.0 PL=0
MOVL C00741 V=800.0 PL=0
MOVL C00742 V=800.0 PL=0
MOVL C00743 V=800.0 PL=0
MOVL C00744 V=800.0 PL=0
MOVL C00745 V=800.0 PL=0
MOVL C00746 V=800.0 PL=0
MOVL C00747 V=800.0 PL=0
MOVL C00748 V=800.0 PL=0
MOVL C00749 V=800.0 PL=0
MOVL C00750 V=800.0 PL=0
MOVL C00751 V=800.0 PL=0
MOVL C00752 V=800.0 PL=0
MOVL C00753 V=800.0 PL=0
MOVL C00754 V=800.0 PL=0
MOVL C00755 V=800.0 PL=0
MOVL C00756 V=800.0 PL=0
MOVL C00757 V=800.0 PL=0
MOVL C00758 V=800.0 PL=0
MOVL C00759 V=800.0 PL=0
MOVL C00760 V=800.0 PL=0
MOVL C00761 V=800.0 PL=0
MOVL C00762 V=800.0 PL=0
MOVL C00763 V=800.0 PL=0
MOVL C00764 V=800.0 PL=0
MOVL C00765 V=800.0 PL=0
MOVL C00766 V=800.0 PL=0
MOVL C00767 V=800.0 PL=0
MOVL C00768 V=800.0 PL=0
MOVL C00769 V=800.0 PL=0
MOVL C00770 V=800.0 PL=0
MOVL C00771 V=800.0 PL=0
MOVL C00772 V=800.0 PL=0
MOVL C00773 V=800.0 PL=0
MOVL C00774 V=800.0 PL=0
MOVL C00775 V=800.0 PL=0
MOVL C00776 V=800.0 PL=0
MOVL C00777 V=800.0 PL=0
MOVL C00778 V=800.0 PL=0
MOVL C00779 V=800.0 PL=0
MOVL C00780 V=800.0 PL=0
MOVL C00781 V=800.0 PL=0
MOVL C00782 V=800.0 PL=0
MOVL C00783 V=800.0 PL=0
MOVL C00784 V=800.0 PL=0
MOVL C00785 V=800.0 PL=0
MOVL C00786 V=800.0 PL=0
MOVL C00787 V=800.0 PL=0
MOVL C00788 V=800.0 PL=0
MOVL C00789 V=800.0 PL=0
MOVL C00790 V=800.0 PL=0
MOVL C00791 V=800.0 PL=0
MOVL C00792 V=800.0 PL=0
MOVL C00793 V=800.0 PL=0
MOVL C00794 V=800.0 PL=0
MOVL C00795 V=800.0 PL=0
MOVL C00796 V=800.0 PL=0
MOVL C00797 V=800.0 PL=0
MOVL C00798 V=800.0 PL=0
MOVL C00799 V=800.0 PL=0
MOVL C00800 V=800.0 PL=0
MOVL C00801 V=800.0 PL=0
MOVL C00802 V=800.0 PL=0
MOVL C00803 V=800.0 PL=0
MOVL C00804 V=800.0 PL=0
MOVL C00805 V=800.0 PL=0
MOVL C00806 V=800.0 PL=0
MOVL C00807 V=800.0 PL=0
MOVL C00808 V=800.0 PL=0
MOVL C00809 V=800.0 PL=0
MOVL C00810 V=800.0 PL=0
MOVL C00811 V=800.0 PL=0
MOVL C00812 V=800.0 PL=0
MOVL C00813 V=800.0 PL=0
MOVL C00814 V=800.0 PL=0
MOVL C00815 V=800.0 PL=0
MOVL C00816 V=800.0 PL=0
MOVL C00817 V=800.0 PL=0
MOVL C00818 V=800.0 PL=0
MOVL C00819 V=800.0 PL=0
MOVL C00820 V=800.0 PL=0
MOVL C00821 V=800.0 PL=0
MOVL C00822 V=800.0 PL=0
MOVL C00823 V=800.0 PL=0
MOVL C00824 V=800.0 PL=0
MOVL C00825 V=800.0 PL=0
MOVL C00826 V=800.0 PL=0
MOVL C00827 V=800.0 PL=0
MOVL C00828 V=800.0 PL=0
MOVL C00829 V=800.0 PL=0
MOVL C00830 V=800.0 PL=0
MOVL C00831 V=800.0 PL=0
MOVL C00832 V=800.0 PL=0
MOVL C00833 V=800.0 PL=0
MOVL C00834 V=800.0 PL=0
MOVL C00835 V=800.0 PL=0
MOVL C00836 V=800.0 PL=0
MOVL C00837 V=800.0 PL=0
MOVL C00838 V=800.0 PL=0
MOVL C00839 V=800.0 PL=0
MOVL C00840 V=800.0 PL=0
MOVL C00841 V=800.0 PL=0
MOVL C00842 V=800.0 PL=0
MOVL C00843 V=800.0 PL=0
MOVL C00844 V=800.0 PL=0
MOVL C00845 V=800.0 PL=0
MOVL C00846 V=800.0 PL=0
MOVL C00847 V=800.0 PL=0
MOVL C00848 V=800.0 PL=0
MOVL C00849 V=800.0 PL=0
MOVL C00850 V=800.0 PL=0
MOVL C00851 V=800.0 PL=0
MOVL C00852 V=800.0 PL=0
MOVL C00853 V=800.0 PL=0
MOVL C00854 V=800.0 PL=0
MOVL C00855 V=800.0 PL=0
MOVL C00856 V=800.0 PL=0
MOVL C00857 V=800.0 PL=0
MOVL C00858 V=800.0 PL=0
MOVL C00859 V=800.0 PL=0
MOVL C00860 V=800.0 PL=0
MOVL C00861 V=800.0 PL=0
MOVL C00862 V=800.0 PL=0
MOVL C00863 V=800.0 PL=0
MOVL C00864 V=800.0 PL=0
MOVL C00865 V=800.0 PL=0
MOVL C00866 V=800.0 PL=0
MOVL C00867 V=800.0 PL=0
MOVL C00868 V=800.0 PL=0
MOVL C00869 V=800.0 PL=0
MOVL C00870 V=800.0 PL=0
MOVL C00871 V=800.0 PL=0
MOVL C00872 V=800.0 PL=0
MOVL C00873 V=800.0 PL=0
MOVL C00874 V=800.0 PL=0
MOVL C00875 V=800.0 PL=0
MOVL C00876 V=800.0 PL=0
MOVL C00877 V=800.0 PL=0
MOVL C00878 V=800.0 PL=0
MOVL C00879 V=800.0 PL=0
MOVL C00880 V=800.0 PL=0
MOVL C00881 V=800.0 PL=0
MOVL C00882 V=800.0 PL=0
MOVL C00883 V=800.0 PL=0
MOVL C00884 V=800.0 PL=0
MOVL C00885 V=800.0 PL=0
MOVL C00886 V=800.0 PL=0
MOVL C00887 V=800.0 PL=0
MOVL C00888 V=800.0 PL=0
MOVL C00889 V=800.0 PL=0
MOVL C00890 V=800.0 PL=0
MOVL C00891 V=800.0 PL=0
MOVL C00892 V=800.0 PL=0
MOVL C00893 V=800.0 PL=0
MOVL C00894 V=800.0 PL=0
MOVL C00895 V=800.0 PL=0
MOVL C00896 V=800.0 PL=0
MOVL C00897 V=800.0 PL=0
MOVL C00898 V=800.0 PL=0
MOVL C00899 V=800.0 PL=0
MOVL C00900 V=800.0 PL=0
MOVL C00901 V=800.0 PL=0
MOVL C00902 V=800.0 PL=0
MOVL C00903 V=800.0 PL=0
MOVL C00904 V=800.0 PL=0
MOVL C00905 V=800.0 PL=0
MOVL C00906 V=800.0 PL=0
MOVL C00907 V=800.0 PL=0
MOVL C00908 V=800.0 PL=0
MOVL C00909 V=800.0 PL=0
MOVL C00910 V=800.0 PL=0
MOVL C00911 V=800.0 PL=0
MOVL C00912 V=800.0 PL=0
MOVL C00913 V=800.0 PL=0
MOVL C00914 V=800.0 PL=0
MOVL C00915 V=800.0 PL=0
MOVL C00916 V=800.0 PL=0
MOVL C00917 V=800.0 PL=0
MOVL C00918 V=800.0 PL=0
MOVL C00919 V=800.0 PL=0
MOVL C00920 V=800.0 PL=0
MOVL C00921 V=800.0 PL=0
MOVL C00922 V=800.0 PL=0
MOVL C00923 V=800.0 PL=0
MOVL C00924 V=800.0 PL=0
MOVL C00925 V=800.0 PL=0
MOVL C00926 V=800.0 PL=0
MOVL C00927 V=800.0 PL=0
MOVL C00928 V=800.0 PL=0
MOVL C00929 V=800.0 PL=0
MOVL C00930 V=800.0 PL=0
MOVL C00931 V=800.0 PL=0
MOVL C00932 V=800.0 PL=0
MOVL C00933 V=800.0 PL=0
MOVL C00934 V=800.0 PL=0
MOVL C00935 V=800.0 PL=0
MOVL C00936 V=800.0 PL=0
MOVL C00937 V=800.0 PL=0
MOVL C00938 V=800.0 PL=0
MOVL C00939 V=800.0 PL=0
MOVL C00940 V=800.0 PL=0
MOVL C00941 V=800.0 PL=0
MOVL C00942 V=800.0 PL=0
MOVL C00943 V=800.0 PL=0
MOVL C00944 V=800.0 PL=0
MOVL C00945 V=800.0 PL=0
MOVL C00946 V=800.0 PL=0
MOVL C00947 V=800.0 PL=0
MOVL C00948 V=800.0 PL=0
MOVL C00949 V=800.0 PL=0
MOVL C00950 V=800.0 PL=0
MOVL C00951 V=800.0 PL=0
MOVL C00952 V=800.0 PL=0
MOVL C00953 V=800.0 PL=0
MOVL C00954 V=800.0 PL=0
MOVL C00955 V=800.0 PL=0
MOVL C00956 V=800.0 PL=0
MOVL C00957 V=800.0 PL=0
MOVL C00958 V=800.0 PL=0
MOVL C00959 V=800.0 PL=0
MOVL C00960 V=800.0 PL=0
MOVL C00961 V=800.0 PL=0
MOVL C00962 V=800.0 PL=0
MOVL C00963 V=800.0 PL=0
MOVL C00964 V=800.0 PL=0
MOVL C00965 V=800.0 PL=0
MOVL C00966 V=800.0 PL=0
MOVL C00967 V=800.0 PL=0
MOVL C00968 V=800.0 PL=0
MOVL C00969 V=800.0 PL=0
MOVL C00970 V=800.0 PL=0
MOVL C00971 V=800.0 PL=0
MOVL C00972 V=800.0 PL=0
MOVL C00973 V=800.0 PL=0
MOVL C00974 V=800.0 PL=0
MOVL C00975 V=800.0 PL=0
MOVL C00976 V=800.0 PL=0
MOVL C00977 V=800.0 PL=0
MOVL C00978 V=800.0 PL=0
MOVL C00979 V=800.0 PL=0
MOVL C00980 V=800.0 PL=0
MOVL C00981 V=800.0 PL=0
MOVL C00982 V=800.0 PL=0
MOVL C00983 V=800.0 PL=0
MOVL C00984 V=800.0 PL=0
MOVL C00985 V=800.0 PL=0
MOVL C00986 V=800.0 PL=0
MOVL C00987 V=800.0 PL=0
MOVL C00988 V=800.0 PL=0
MOVL C00989 V=800.0 PL=0
MOVL C00990 V=800.0 PL=0
MOVL C00991 V=800.0 PL=0
MOVL C00992 V=800.0 PL=0
MOVL C00993 V=800.0 PL=0
MOVL C00994 V=800.0 PL=0
MOVL C00995 V=800.0 PL=0
MOVL C00996 V=800.0 PL=0
MOVL C00997 V=800.0 PL=0
MOVL C00998 V=800.0 PL=0
MOVL C00999 V=800.0 PL=0
MOVL C01000 V=800.0 PL=0
MOVL C01001 V=800.0 PL=0
MOVL C01002 V=800.0 PL=0
MOVL C01003 V=800.0 PL=0
MOVL C01004 V=800.0 PL=0
MOVL C01005 V=800.0 PL=0
MOVL C01006 V=800.0 PL=0
MOVL C01007 V=800.0 PL=0
MOVL C01008 V=800.0 PL=0
MOVL C01009 V=800.0 PL=0
MOVL C01010 V=800.0 PL=0
MOVL C01011 V=800.0 PL=0
MOVL C01012 V=800.0 PL=0
MOVL C01013 V=800.0 PL=0
MOVL C01014 V=800.0 PL=0
MOVL C01015 V=800.0 PL=0
MOVL C01016 V=800.0 PL=0
MOVL C01017 V=800.0 PL=0
MOVL C01018 V=800.0 PL=0
MOVL C01019 V=800.0 PL=0
MOVL C01020 V=800.0 PL=0
MOVL C01021 V=800.0 PL=0
MOVL C01022 V=800.0 PL=0
MOVL C01023 V=800.0 PL=0
MOVL C01024 V=800.0 PL=0
MOVL C01025 V=800.0 PL=0
MOVL C01026 V=800.0 PL=0
MOVL C01027 V=800.0 PL=0
MOVL C01028 V=800.0 PL=0
MOVL C01029 V=800.0 PL=0
MOVL C01030 V=800.0 PL=0
MOVL C01031 V=800.0 PL=0
MOVL C01032 V=800.0 PL=0
MOVL C01033 V=800.0 PL=0
MOVL C01034 V=800.0 PL=0
MOVL C01035 V=800.0 PL=0
MOVL C01036 V=800.0 PL=0
MOVL C01037 V=800.0 PL=0
MOVL C01038 V=800.0 PL=0
MOVL C01039 V=800.0 PL=0
MOVL C01040 V=800.0 PL=0
MOVL C01041 V=800.0 PL=0
MOVL C01042 V=800.0 PL=0
MOVL C01043 V=800.0 PL=0
MOVL C01044 V=800.0 PL=0
MOVL C01045 V=800.0 PL=0
MOVL C01046 V=800.0 PL=0
MOVL C01047 V=800.0 PL=0
MOVL C01048 V=800.0 PL=0
MOVL C01049 V=800.0 PL=0
MOVL C01050 V=800.0 PL=0
MOVL C01051 V=800.0 PL=0
MOVL C01052 V=800.0 PL=0
MOVL C01053 V=800.0 PL=0
MOVL C01054 V=800.0 PL=0
MOVL C01055 V=800.0 PL=0
MOVL C01056 V=800.0 PL=0
MOVL C01057 V=800.0 PL=0
MOVL C01058 V=800.0 PL=0
MOVL C01059 V=800.0 PL=0
MOVL C01060 V=800.0 PL=0
MOVL C01061 V=800.0 PL=0
MOVL C01062 V=800.0 PL=0
MOVL C01063 V=800.0 PL=0
MOVL C01064 V=800.0 PL=0
MOVL C01065 V=800.0 PL=0
MOVL C01066 V=800.0 PL=0
MOVL C01067 V=800.0 PL=0
MOVL C01068 V=800.0 PL=0
MOVL C01069 V=800.0 PL=0
MOVL C01070 V=800.0 PL=0
MOVL C01071 V=800.0 PL=0
MOVL C01072 V=800.0 PL=0
MOVL C01073 V=800.0 PL=0
MOVL C01074 V=800.0 PL=0
MOVL C01075 V=800.0 PL=0
MOVL C01076 V=800.0 PL=0
MOVL C01077 V=800.0 PL=0
MOVL C01078 V=800.0 PL=0
MOVL C01079 V=800.0 PL=0
MOVL C01080 V=800.0 PL=0
MOVL C01081 V=800.0 PL=0
MOVL C01082 V=800.0 PL=0
MOVL C01083 V=800.0 PL=0
MOVL C01084 V=800.0 PL=0
MOVL C01085 V=800.0 PL=0
MOVL C01086 V=800.0 PL=0
MOVL C01087 V=800.0 PL=0
MOVL C01088 V=800.0 PL=0
MOVL C01089 V=800.0 PL=0
MOVL C01090 V=800.0 PL=0
MOVL C01091 V=800.0 PL=0
MOVL C01092 V=800.0 PL=0
MOVL C01093 V=800.0 PL=0
MOVL C01094 V=800.0 PL=0
MOVL C01095 V=800.0 PL=0
MOVL C01096 V=800.0 PL=0
MOVL C01097 V=800.0 PL=0
MOVL C01098 V=800.0 PL=0
MOVL C01099 V=800.0 PL=0
MOVL C01100 V=800.0 PL=0
MOVL C01101 V=800.0 PL=0
MOVL C01102 V=800.0 PL=0
MOVL C01103 V=800.0 PL=0
MOVL C01104 V=800.0 PL=0
MOVL C01105 V=800.0 PL=0
MOVL C01106 V=800.0 PL=0
MOVL C01107 V=800.0 PL=0
MOVL C01108 V=800.0 PL=0
MOVL C01109 V=800.0 PL=0
MOVL C01110 V=800.0 PL=0
MOVL C01111 V=800.0 PL=0
MOVL C01112 V=800.0 PL=0
MOVL C01113 V=800.0 PL=0
MOVL C01114 V=800.0 PL=0
MOVL C01115 V=800.0 PL=0
MOVL C01116 V=800.0 PL=0
MOVL C01117 V=800.0 PL=0
MOVL C01118 V=800.0 PL=0
MOVL C01119 V=800.0 PL=0
MOVL C01120 V=800.0 PL=0
MOVL C01121 V=800.0 PL=0
MOVL C01122 V=800.0 PL=0
MOVL C01123 V=800.0 PL=0
MOVL C01124 V=800.0 PL=0
MOVL C01125 V=800.0 PL=0
MOVL C01126 V=800.0 PL=0
MOVL C01127 V=800.0 PL=0
MOVL C01128 V=800.0 PL=0
MOVL C01129 V=800.0 PL=0
MOVL C01130 V=800.0 PL=0
MOVL C01131 V=800.0 PL=0
MOVL C01132 V=800.0 PL=0
MOVL C01133 V=800.0 PL=0
MOVL C01134 V=800.0 PL=0
MOVL C01135 V=800.0 PL=0
MOVL C01136 V=800.0 PL=0
MOVL C01137 V=800.0 PL=0
MOVL C01138 V=800.0 PL=0
MOVL C01139 V=800.0 PL=0
MOVL C01140 V=800.0 PL=0
MOVL C01141 V=800.0 PL=0
MOVL C01142 V=800.0 PL=0
MOVL C01143 V=800.0 PL=0
MOVL C01144 V=800.0 PL=0
MOVL C01145 V=800.0 PL=0
MOVL C01146 V=800.0 PL=0
MOVL C01147 V=800.0 PL=0
MOVL C01148 V=800.0 PL=0
MOVL C01149 V=800.0 PL=0
MOVL C01150 V=800.0 PL=0
MOVL C01151 V=800.0 PL=0
MOVL C01152 V=800.0 PL=0
MOVL C01153 V=800.0 PL=0
MOVL C01154 V=800.0 PL=0
MOVL C01155 V=800.0 PL=0
MOVL C01156 V=800.0 PL=0
MOVL C01157 V=800.0 PL=0
MOVL C01158 V=800.0 PL=0
MOVL C01159 V=800.0 PL=0
MOVL C01160 V=800.0 PL=0
MOVL C01161 V=800.0 PL=0
MOVL C01162 V=800.0 PL=0
MOVL C01163 V=800.0 PL=0
MOVL C01164 V=800.0 PL=0
MOVL C01165 V=800.0 PL=0
MOVL C01166 V=800.0 PL=0
MOVL C01167 V=800.0 PL=0
MOVL C01168 V=800.0 PL=0
MOVL C01169 V=800.0 PL=0
MOVL C01170 V=800.0 PL=0
MOVL C01171 V=800.0 PL=0
MOVL C01172 V=800.0 PL=0
MOVL C01173 V=800.0 PL=0
MOVL C01174 V=800.0 PL=0
MOVL C01175 V=800.0 PL=0
MOVL C01176 V=800.0 PL=0
MOVL C01177 V=800.0 PL=0
MOVL C01178 V=800.0 PL=0
MOVL C01179 V=800.0 PL=0
MOVL C01180 V=800.0 PL=0
MOVL C01181 V=800.0 PL=0
MOVL C01182 V=800.0 PL=0
MOVL C01183 V=800.0 PL=0
MOVL C01184 V=800.0 PL=0
MOVL C01185 V=800.0 PL=0
MOVL C01186 V=800.0 PL=0
MOVL C01187 V=800.0 PL=0
MOVL C01188 V=800.0 PL=0
MOVL C01189 V=800.0 PL=0
MOVL C01190 V=800.0 PL=0
MOVL C01191 V=800.0 PL=0
MOVL C01192 V=800.0 PL=0
MOVL C01193 V=800.0 PL=0
MOVL C01194 V=800.0 PL=0
MOVL C01195 V=800.0 PL=0
MOVL C01196 V=800.0 PL=0
MOVL C01197 V=800.0 PL=0
MOVL C01198 V=800.0 PL=0
MOVL C01199 V=800.0 PL=0
MOVL C01200 V=800.0 PL=0
MOVL C01201 V=800.0 PL=0
MOVL C01202 V=800.0 PL=0
MOVL C01203 V=800.0 PL=0
MOVL C01204 V=800.0 PL=0
MOVL C01205 V=800.0 PL=0
MOVL C01206 V=800.0 PL=0
MOVL C01207 V=800.0 PL=0
MOVL C01208 V=800.0 PL=0
MOVL C01209 V=800.0 PL=0
MOVL C01210 V=800.0 PL=0
MOVL C01211 V=800.0 PL=0
MOVL C01212 V=800.0 PL=0
MOVL C01213 V=800.0 PL=0
MOVL C01214 V=800.0 PL=0
MOVL C01215 V=800.0 PL=0
MOVL C01216 V=800.0 PL=0
MOVL C01217 V=800.0 PL=0
MOVL C01218 V=800.0 PL=0
MOVL C01219 V=800.0 PL=0
MOVL C01220 V=800.0 PL=0
MOVL C01221 V=800.0 PL=0
MOVL C01222 V=800.0 PL=0
MOVL C01223 V=800.0 PL=0
MOVL C01224 V=800.0 PL=0
MOVL C01225 V=800.0 PL=0
MOVL C01226 V=800.0 PL=0
MOVL C01227 V=800.0 PL=0
MOVL C01228 V=800.0 PL=0
MOVL C01229 V=800.0 PL=0
MOVL C01230 V=800.0 PL=0
MOVL C01231 V=800.0 PL=0
MOVL C01232 V=800.0 PL=0
MOVL C01233 V=800.0 PL=0
MOVL C01234 V=800.0 PL=0
MOVL C01235 V=800.0 PL=0
MOVL C01236 V=800.0 PL=0
MOVL C01237 V=800.0 PL=0
MOVL C01238 V=800.0 PL=0
MOVL C01239 V=800.0 PL=0
MOVL C01240 V=800.0 PL=0
MOVL C01241 V=800.0 PL=0
MOVL C01242 V=800.0 PL=0
MOVL C01243 V=800.0 PL=0
MOVL C01244 V=800.0 PL=0
MOVL C01245 V=800.0 PL=0
MOVL C01246 V=800.0 PL=0
MOVL C01247 V=800.0 PL=0
MOVL C01248 V=800.0 PL=0
MOVL C01249 V=800.0 PL=0
MOVL C01250 V=800.0 PL=0
MOVL C01251 V=800.0 PL=0
MOVL C01252 V=800.0 PL=0
MOVL C01253 V=800.0 PL=0
MOVL C01254 V=800.0 PL=0
MOVL C01255 V=800.0 PL=0
MOVL C01256 V=800.0 PL=0
MOVL C01257 V=800.0 PL=0
MOVL C01258 V=800.0 PL=0
MOVL C01259 V=800.0 PL=0
MOVL C01260 V=800.0 PL=0
MOVL C01261 V=800.0 PL=0
MOVL C01262 V=800.0 PL=0
MOVL C01263 V=800.0 PL=0
MOVL C01264 V=800.0 PL=0
MOVL C01265 V=800.0 PL=0
MOVL C01266 V=800.0 PL=0
MOVL C01267 V=800.0 PL=0
MOVL C01268 V=800.0 PL=0
MOVL C01269 V=800.0 PL=0
MOVL C01270 V=800.0 PL=0
MOVL C01271 V=800.0 PL=0
MOVL C01272 V=800.0 PL=0
MOVL C01273 V=800.0 PL=0
MOVL C01274 V=800.0 PL=0
MOVL C01275 V=800.0 PL=0
MOVL C01276 V=800.0 PL=0
MOVL C01277 V=800.0 PL=0
MOVL C01278 V=800.0 PL=0
MOVL C01279 V=800.0 PL=0
MOVL C01280 V=800.0 PL=0
MOVL C01281 V=800.0 PL=0
MOVL C01282 V=800.0 PL=0
MOVL C01283 V=800.0 PL=0
MOVL C01284 V=800.0 PL=0
MOVL C01285 V=800.0 PL=0
MOVL C01286 V=800.0 PL=0
MOVL C01287 V=800.0 PL=0
MOVL C01288 V=800.0 PL=0
MOVL C01289 V=800.0 PL=0
MOVL C01290 V=800.0 PL=0
MOVL C01291 V=800.0 PL=0
MOVL C01292 V=800.0 PL=0
MOVL C01293 V=800.0 PL=0
MOVL C01294 V=800.0 PL=0
MOVL C01295 V=800.0 PL=0
MOVL C01296 V=800.0 PL=0
MOVL C01297 V=800.0 PL=0
MOVL C01298 V=800.0 PL=0
MOVL C01299 V=800.0 PL=0
MOVL C01300 V=800.0 PL=0
MOVL C01301 V=800.0 PL=0
MOVL C01302 V=800.0 PL=0
MOVL C01303 V=800.0 PL=0
MOVL C01304 V=800.0 PL=0
MOVL C01305 V=800.0 PL=0
MOVL C01306 V=800.0 PL=0
MOVL C01307 V=800.0 PL=0
MOVL C01308 V=800.0 PL=0
MOVL C01309 V=800.0 PL=0
MOVL C01310 V=800.0 PL=0
MOVL C01311 V=800.0 PL=0
MOVL C01312 V=800.0 PL=0
MOVL C01313 V=800.0 PL=0
MOVL C01314 V=800.0 PL=0
MOVL C01315 V=800.0 PL=0
MOVL C01316 V=800.0 PL=0
MOVL C01317 V=800.0 PL=0
MOVL C01318 V=800.0 PL=0
MOVL C01319 V=800.0 PL=0
MOVL C01320 V=800.0 PL=0
MOVL C01321 V=800.0 PL=0
MOVL C01322 V=800.0 PL=0
MOVL C01323 V=800.0 PL=0
MOVL C01324 V=800.0 PL=0
MOVL C01325 V=800.0 PL=0
MOVL C01326 V=800.0 PL=0
MOVL C01327 V=800.0 PL=0
MOVL C01328 V=800.0 PL=0
MOVL C01329 V=800.0 PL=0
MOVL C01330 V=800.0 PL=0
MOVL C01331 V=800.0 PL=0
MOVL C01332 V=800.0 PL=0
MOVL C01333 V=800.0 PL=0
MOVL C01334 V=800.0 PL=0
MOVL C01335 V=800.0 PL=0
MOVL C01336 V=800.0 PL=0
MOVL C01337 V=800.0 PL=0
MOVL C01338 V=800.0 PL=0
MOVL C01339 V=800.0 PL=0
MOVL C01340 V=800.0 PL=0
MOVL C01341 V=800.0 PL=0
MOVL C01342 V=800.0 PL=0
MOVL C01343 V=800.0 PL=0
MOVL C01344 V=800.0 PL=0
MOVL C01345 V=800.0 PL=0
MOVL C01346 V=800.0 PL=0
MOVL C01347 V=800.0 PL=0
MOVL C01348 V=800.0 PL=0
MOVL C01349 V=800.0 PL=0
MOVL C01350 V=800.0 PL=0
MOVL C01351 V=800.0 PL=0
MOVL C01352 V=800.0 PL=0
MOVL C01353 V=800.0 PL=0
MOVL C01354 V=800.0 PL=0
MOVL C01355 V=800.0 PL=0
MOVL C01356 V=800.0 PL=0
MOVL C01357 V=800.0 PL=0
MOVL C01358 V=800.0 PL=0
MOVL C01359 V=800.0 PL=0
MOVL C01360 V=800.0 PL=0
MOVL C01361 V=800.0 PL=0
MOVL C01362 V=800.0 PL=0
MOVL C01363 V=800.0 PL=0
MOVL C01364 V=800.0 PL=0
MOVL C01365 V=800.0 PL=0
MOVL C01366 V=800.0 PL=0
MOVL C01367 V=800.0 PL=0
MOVL C01368 V=800.0 PL=0
MOVL C01369 V=800.0 PL=0
MOVL C01370 V=800.0 PL=0
MOVL C01371 V=800.0 PL=0
MOVL C01372 V=800.0 PL=0
MOVL C01373 V=800.0 PL=0
MOVL C01374 V=800.0 PL=0
MOVL C01375 V=800.0 PL=0
MOVL C01376 V=800.0 PL=0
MOVL C01377 V=800.0 PL=0
MOVL C01378 V=800.0 PL=0
MOVL C01379 V=800.0 PL=0
MOVL C01380 V=800.0 PL=0
MOVL C01381 V=800.0 PL=0
MOVL C01382 V=800.0 PL=0
MOVL C01383 V=800.0 PL=0
MOVL C01384 V=800.0 PL=0
MOVL C01385 V=800.0 PL=0
MOVL C01386 V=800.0 PL=0
MOVL C01387 V=800.0 PL=0
MOVL C01388 V=800.0 PL=0
MOVL C01389 V=800.0 PL=0
MOVL C01390 V=800.0 PL=0
MOVL C01391 V=800.0 PL=0
MOVL C01392 V=800.0 PL=0
MOVL C01393 V=800.0 PL=0
MOVL C01394 V=800.0 PL=0
MOVL C01395 V=800.0 PL=0
MOVL C01396 V=800.0 PL=0
MOVL C01397 V=800.0 PL=0
MOVL C01398 V=800.0 PL=0
MOVL C01399 V=800.0 PL=0
MOVL C01400 V=800.0 PL=0
MOVL C01401 V=800.0 PL=0
MOVL C01402 V=800.0 PL=0
MOVL C01403 V=800.0 PL=0
MOVL C01404 V=800.0 PL=0
MOVL C01405 V=800.0 PL=0
MOVL C01406 V=800.0 PL=0
MOVL C01407 V=800.0 PL=0
MOVL C01408 V=800.0 PL=0
MOVL C01409 V=800.0 PL=0
MOVL C01410 V=800.0 PL=0
MOVL C01411 V=800.0 PL=0
MOVL C01412 V=800.0 PL=0
MOVL C01413 V=800.0 PL=0
MOVL C01414 V=800.0 PL=0
MOVL C01415 V=800.0 PL=0
MOVL C01416 V=800.0 PL=0
MOVL C01417 V=800.0 PL=0
MOVL C01418 V=800.0 PL=0
MOVL C01419 V=800.0 PL=0
MOVL C01420 V=800.0 PL=0
MOVL C01421 V=800.0 PL=0
MOVL C01422 V=800.0 PL=0
MOVL C01423 V=800.0 PL=0
MOVL C01424 V=800.0 PL=0
MOVL C01425 V=800.0 PL=0
MOVL C01426 V=800.0 PL=0
MOVL C01427 V=800.0 PL=0
MOVL C01428 V=800.0 PL=0
MOVL C01429 V=800.0 PL=0
MOVL C01430 V=800.0 PL=0
MOVL C01431 V=800.0 PL=0
MOVL C01432 V=800.0 PL=0
MOVL C01433 V=800.0 PL=0
MOVL C01434 V=800.0 PL=0
MOVL C01435 V=800.0 PL=0
MOVL C01436 V=800.0 PL=0
MOVL C01437 V=800.0 PL=0
MOVL C01438 V=800.0 PL=0
MOVL C01439 V=800.0 PL=0
MOVL C01440 V=800.0 PL=0
MOVL C01441 V=800.0 PL=0
MOVL C01442 V=800.0 PL=0
MOVL C01443 V=800.0 PL=0
MOVL C01444 V=800.0 PL=0
MOVL C01445 V=800.0 PL=0
MOVL C01446 V=800.0 PL=0
MOVL C01447 V=800.0 PL=0
MOVL C01448 V=800.0 PL=0
MOVL C01449 V=800.0 PL=0
MOVL C01450 V=800.0 PL=0
MOVL C01451 V=800.0 PL=0
MOVL C01452 V=800.0 PL=0
MOVL C01453 V=800.0 PL=0
MOVL C01454 V=800.0 PL=0
MOVL C01455 V=800.0 PL=0
MOVL C01456 V=800.0 PL=0
MOVL C01457 V=800.0 PL=0
MOVL C01458 V=800.0 PL=0
MOVL C01459 V=800.0 PL=0
MOVL C01460 V=800.0 PL=0
MOVL C01461 V=800.0 PL=0
MOVL C01462 V=800.0 PL=0
MOVL C01463 V=800.0 PL=0
MOVL C01464 V=800.0 PL=0
MOVL C01465 V=800.0 PL=0
MOVL C01466 V=800.0 PL=0
MOVL C01467 V=800.0 PL=0
MOVL C01468 V=800.0 PL=0
MOVL C01469 V=800.0 PL=0
MOVL C01470 V=800.0 PL=0
MOVL C01471 V=800.0 PL=0
MOVL C01472 V=800.0 PL=0
MOVL C01473 V=800.0 PL=0
MOVL C01474 V=800.0 PL=0
MOVL C01475 V=800.0 PL=0
MOVL C01476 V=800.0 PL=0
MOVL C01477 V=800.0 PL=0
MOVL C01478 V=800.0 PL=0
MOVL C01479 V=800.0 PL=0
MOVL C01480 V=800.0 PL=0
MOVL C01481 V=800.0 PL=0
MOVL C01482 V=800.0 PL=0
MOVL C01483 V=800.0 PL=0
MOVL C01484 V=800.0 PL=0
MOVL C01485 V=800.0 PL=0
MOVL C01486 V=800.0 PL=0
MOVL C01487 V=800.0 PL=0
MOVL C01488 V=800.0 PL=0
MOVL C01489 V=800.0 PL=0
MOVL C01490 V=800.0 PL=0
MOVL C01491 V=800.0 PL=0
MOVL C01492 V=800.0 PL=0
MOVL C01493 V=800.0 PL=0
MOVL C01494 V=800.0 PL=0
MOVL C01495 V=800.0 PL=0
MOVL C01496 V=800.0 PL=0
MOVL C01497 V=800.0 PL=0
MOVL C01498 V=800.0 PL=0
MOVL C01499 V=800.0 PL=0
MOVL C01500 V=800.0 PL=0
MOVL C01501 V=800.0 PL=0
MOVL C01502 V=800.0 PL=0
MOVL C01503 V=800.0 PL=0
MOVL C01504 V=800.0 PL=0
MOVL C01505 V=800.0 PL=0
MOVL C01506 V=800.0 PL=0
MOVL C01507 V=800.0 PL=0
MOVL C01508 V=800.0 PL=0
MOVL C01509 V=800.0 PL=0
MOVL C01510 V=800.0 PL=0
MOVL C01511 V=800.0 PL=0
MOVL C01512 V=800.0 PL=0
MOVL C01513 V=800.0 PL=0
MOVL C01514 V=800.0 PL=0
MOVL C01515 V=800.0 PL=0
MOVL C01516 V=800.0 PL=0
MOVL C01517 V=800.0 PL=0
MOVL C01518 V=800.0 PL=0
MOVL C01519 V=800.0 PL=0
MOVL C01520 V=800.0 PL=0
MOVL C01521 V=800.0 PL=0
MOVL C01522 V=800.0 PL=0
MOVL C01523 V=800.0 PL=0
MOVL C01524 V=800.0 PL=0
MOVL C01525 V=800.0 PL=0
MOVL C01526 V=800.0 PL=0
MOVL C01527 V=800.0 PL=0
MOVL C01528 V=800.0 PL=0
MOVL C01529 V=800.0 PL=0
MOVL C01530 V=800.0 PL=0
MOVL C01531 V=800.0 PL=0
MOVL C01532 V=800.0 PL=0
MOVL C01533 V=800.0 PL=0
MOVL C01534 V=800.0 PL=0
MOVL C01535 V=800.0 PL=0
MOVL C01536 V=800.0 PL=0
MOVL C01537 V=800.0 PL=0
MOVL C01538 V=800.0 PL=0
MOVL C01539 V=800.0 PL=0
MOVL C01540 V=800.0 PL=0
MOVL C01541 V=800.0 PL=0
MOVL C01542 V=800.0 PL=0
MOVL C01543 V=800.0 PL=0
MOVL C01544 V=800.0 PL=0
MOVL C01545 V=800.0 PL=0
MOVL C01546 V=800.0 PL=0
MOVL C01547 V=800.0 PL=0
MOVL C01548 V=800.0 PL=0
MOVL C01549 V=800.0 PL=0
MOVL C01550 V=800.0 PL=0
MOVL C01551 V=800.0 PL=0
MOVL C01552 V=800.0 PL=0
MOVL C01553 V=800.0 PL=0
MOVL C01554 V=800.0 PL=0
MOVL C01555 V=800.0 PL=0
MOVL C01556 V=800.0 PL=0
MOVL C01557 V=800.0 PL=0
MOVL C01558 V=800.0 PL=0
MOVL C01559 V=800.0 PL=0
MOVL C01560 V=800.0 PL=0
MOVL C01561 V=800.0 PL=0
MOVL C01562 V=800.0 PL=0
MOVL C01563 V=800.0 PL=0
MOVL C01564 V=800.0 PL=0
MOVL C01565 V=800.0 PL=0
MOVL C01566 V=800.0 PL=0
MOVL C01567 V=800.0 PL=0
MOVL C01568 V=800.0 PL=0
MOVL C01569 V=800.0 PL=0
MOVL C01570 V=800.0 PL=0
MOVL C01571 V=800.0 PL=0
MOVL C01572 V=800.0 PL=0
MOVL C01573 V=800.0 PL=0
MOVL C01574 V=800.0 PL=0
MOVL C01575 V=800.0 PL=0
MOVL C01576 V=800.0 PL=0
MOVL C01577 V=800.0 PL=0
MOVL C01578 V=800.0 PL=0
MOVL C01579 V=800.0 PL=0
MOVL C01580 V=800.0 PL=0
MOVL C01581 V=800.0 PL=0
MOVL C01582 V=800.0 PL=0
MOVL C01583 V=800.0 PL=0
MOVL C01584 V=800.0 PL=0
MOVL C01585 V=800.0 PL=0
MOVL C01586 V=800.0 PL=0
MOVL C01587 V=800.0 PL=0
MOVL C01588 V=800.0 PL=0
MOVL C01589 V=800.0 PL=0
MOVL C01590 V=800.0 PL=0
MOVL C01591 V=800.0 PL=0
MOVL C01592 V=800.0 PL=0
MOVL C01593 V=800.0 PL=0
MOVL C01594 V=800.0 PL=0
MOVL C01595 V=800.0 PL=0
MOVL C01596 V=800.0 PL=0
MOVL C01597 V=800.0 PL=0
MOVL C01598 V=800.0 PL=0
MOVL C01599 V=800.0 PL=0
MOVL C01600 V=800.0 PL=0
MOVL C01601 V=800.0 PL=0
MOVL C01602 V=800.0 PL=0
MOVL C01603 V=800.0 PL=0
MOVL C01604 V=800.0 PL=0
MOVL C01605 V=800.0 PL=0
MOVL C01606 V=800.0 PL=0
MOVL C01607 V=800.0 PL=0
MOVL C01608 V=800.0 PL=0
MOVL C01609 V=800.0 PL=0
MOVL C01610 V=800.0 PL=0
MOVL C01611 V=800.0 PL=0
MOVL C01612 V=800.0 PL=0
MOVL C01613 V=800.0 PL=0
MOVL C01614 V=800.0 PL=0
MOVL C01615 V=800.0 PL=0
MOVL C01616 V=800.0 PL=0
MOVL C01617 V=800.0 PL=0
MOVL C01618 V=800.0 PL=0
MOVL C01619 V=800.0 PL=0
MOVL C01620 V=800.0 PL=0
MOVL C01621 V=800.0 PL=0
MOVL C01622 V=800.0 PL=0
MOVL C01623 V=800.0 PL=0
MOVL C01624 V=800.0 PL=0
MOVL C01625 V=800.0 PL=0
MOVL C01626 V=800.0 PL=0
MOVL C01627 V=800.0 PL=0
MOVL C01628 V=800.0 PL=0
MOVL C01629 V=800.0 PL=0
MOVL C01630 V=800.0 PL=0
MOVL C01631 V=800.0 PL=0
MOVL C01632 V=800.0 PL=0
MOVL C01633 V=800.0 PL=0
MOVL C01634 V=800.0 PL=0
MOVL C01635 V=800.0 PL=0
MOVL C01636 V=800.0 PL=0
MOVL C01637 V=800.0 PL=0
MOVL C01638 V=800.0 PL=0
MOVL C01639 V=800.0 PL=0
MOVL C01640 V=800.0 PL=0
MOVL C01641 V=800.0 PL=0
MOVL C01642 V=800.0 PL=0
MOVL C01643 V=800.0 PL=0
MOVL C01644 V=800.0 PL=0
MOVL C01645 V=800.0 PL=0
MOVL C01646 V=800.0 PL=0
MOVL C01647 V=800.0 PL=0
MOVL C01648 V=800.0 PL=0
MOVL C01649 V=800.0 PL=0
MOVL C01650 V=800.0 PL=0
MOVL C01651 V=800.0 PL=0
MOVL C01652 V=800.0 PL=0
MOVL C01653 V=800.0 PL=0
MOVL C01654 V=800.0 PL=0
MOVL C01655 V=800.0 PL=0
MOVL C01656 V=800.0 PL=0
MOVL C01657 V=800.0 PL=0
MOVL C01658 V=800.0 PL=0
MOVL C01659 V=800.0 PL=0
MOVL C01660 V=800.0 PL=0
MOVL C01661 V=800.0 PL=0
MOVL C01662 V=800.0 PL=0
MOVL C01663 V=800.0 PL=0
MOVL C01664 V=800.0 PL=0
MOVL C01665 V=800.0 PL=0
MOVL C01666 V=800.0 PL=0
MOVL C01667 V=800.0 PL=0
MOVL C01668 V=800.0 PL=0
MOVL C01669 V=800.0 PL=0
MOVL C01670 V=800.0 PL=0
MOVL C01671 V=800.0 PL=0
MOVL C01672 V=800.0 PL=0
MOVL C01673 V=800.0 PL=0
MOVL C01674 V=800.0 PL=0
MOVL C01675 V=800.0 PL=0
MOVL C01676 V=800.0 PL=0
MOVL C01677 V=800.0 PL=0
MOVL C01678 V=800.0 PL=0
MOVL C01679 V=800.0 PL=0
MOVL C01680 V=800.0 PL=0
MOVL C01681 V=800.0 PL=0
MOVL C01682 V=800.0 PL=0
MOVL C01683 V=800.0 PL=0
MOVL C01684 V=800.0 PL=0
MOVL C01685 V=800.0 PL=0
MOVL C01686 V=800.0 PL=0
MOVL C01687 V=800.0 PL=0
MOVL C01688 V=800.0 PL=0
MOVL C01689 V=800.0 PL=0
MOVL C01690 V=800.0 PL=0
MOVL C01691 V=800.0 PL=0
MOVL C01692 V=800.0 PL=0
MOVL C01693 V=800.0 PL=0
MOVL C01694 V=800.0 PL=0
MOVL C01695 V=800.0 PL=0
MOVL C01696 V=800.0 PL=0
MOVL C01697 V=800.0 PL=0
MOVL C01698 V=800.0 PL=0
MOVL C01699 V=800.0 PL=0
MOVL C01700 V=800.0 PL=0
MOVL C01701 V=800.0 PL=0
MOVL C01702 V=800.0 PL=0
MOVL C01703 V=800.0 PL=0
MOVL C01704 V=800.0 PL=0
MOVL C01705 V=800.0 PL=0
MOVL C01706 V=800.0 PL=0
MOVL C01707 V=800.0 PL=0
MOVL C01708 V=800.0 PL=0
MOVL C01709 V=800.0 PL=0
MOVL C01710 V=800.0 PL=0
MOVL C01711 V=800.0 PL=0
MOVL C01712 V=800.0 PL=0
MOVL C01713 V=800.0 PL=0
MOVL C01714 V=800.0 PL=0
MOVL C01715 V=800.0 PL=0
MOVL C01716 V=800.0 PL=0
MOVL C01717 V=800.0 PL=0
MOVL C01718 V=800.0 PL=0
MOVL C01719 V=800.0 PL=0
MOVL C01720 V=800.0 PL=0
MOVL C01721 V=800.0 PL=0
MOVL C01722 V=800.0 PL=0
MOVL C01723 V=800.0 PL=0
MOVL C01724 V=800.0 PL=0
MOVL C01725 V=800.0 PL=0
MOVL C01726 V=800.0 PL=0
MOVL C01727 V=800.0 PL=0
MOVL C01728 V=800.0 PL=0
MOVL C01729 V=800.0 PL=0
MOVL C01730 V=800.0 PL=0
MOVL C01731 V=800.0 PL=0
MOVL C01732 V=800.0 PL=0
MOVL C01733 V=800.0 PL=0
MOVL C01734 V=800.0 PL=0
MOVL C01735 V=800.0 PL=0
MOVL C01736 V=800.0 PL=0
MOVL C01737 V=800.0 PL=0
MOVL C01738 V=800.0 PL=0
MOVL C01739 V=800.0 PL=0
MOVL C01740 V=800.0 PL=0
MOVL C01741 V=800.0 PL=0
MOVL C01742 V=800.0 PL=0
MOVL C01743 V=800.0 PL=0
MOVL C01744 V=800.0 PL=0
MOVL C01745 V=800.0 PL=0
MOVL C01746 V=800.0 PL=0
MOVL C01747 V=800.0 PL=0
MOVL C01748 V=800.0 PL=0
MOVL C01749 V=800.0 PL=0
MOVL C01750 V=800.0 PL=0
MOVL C01751 V=800.0 PL=0
MOVL C01752 V=800.0 PL=0
MOVL C01753 V=800.0 PL=0
MOVL C01754 V=800.0 PL=0
MOVL C01755 V=800.0 PL=0
MOVL C01756 V=800.0 PL=0
MOVL C01757 V=800.0 PL=0
MOVL C01758 V=800.0 PL=0
MOVL C01759 V=800.0 PL=0
MOVL C01760 V=800.0 PL=0
MOVL C01761 V=800.0 PL=0
MOVL C01762 V=800.0 PL=0
MOVL C01763 V=800.0 PL=0
MOVL C01764 V=800.0 PL=0
MOVL C01765 V=800.0 PL=0
MOVL C01766 V=800.0 PL=0
MOVL C01767 V=800.0 PL=0
MOVL C01768 V=800.0 PL=0
MOVL C01769 V=800.0 PL=0
MOVL C01770 V=800.0 PL=0
MOVL C01771 V=800.0 PL=0
MOVL C01772 V=800.0 PL=0
MOVL C01773 V=800.0 PL=0
MOVL C01774 V=800.0 PL=0
MOVL C01775 V=800.0 PL=0
MOVL C01776 V=800.0 PL=0
MOVL C01777 V=800.0 PL=0
MOVL C01778 V=800.0 PL=0
MOVL C01779 V=800.0 PL=0
MOVL C01780 V=800.0 PL=0
MOVL C01781 V=800.0 PL=0
MOVL C01782 V=800.0 PL=0
MOVL C01783 V=800.0 PL=0
MOVL C01784 V=800.0 PL=0
MOVL C01785 V=800.0 PL=0
MOVL C01786 V=800.0 PL=0
MOVL C01787 V=800.0 PL=0
MOVL C01788 V=800.0 PL=0
MOVL C01789 V=800.0 PL=0
MOVL C01790 V=800.0 PL=0
MOVL C01791 V=800.0 PL=0
MOVL C01792 V=800.0 PL=0
MOVL C01793 V=800.0 PL=0
MOVL C01794 V=800.0 PL=0
MOVL C01795 V=800.0 PL=0
MOVL C01796 V=800.0 PL=0
MOVL C01797 V=800.0 PL=0
MOVL C01798 V=800.0 PL=0
MOVL C01799 V=800.0 PL=0
MOVL C01800 V=800.0 PL=0
MOVL C01801 V=800.0 PL=0
MOVL C01802 V=800.0 PL=0
MOVL C01803 V=800.0 PL=0
MOVL C01804 V=800.0 PL=0
MOVL C01805 V=800.0 PL=0
MOVL C01806 V=800.0 PL=0
MOVL C01807 V=800.0 PL=0
MOVL C01808 V=800.0 PL=0
MOVL C01809 V=800.0 PL=0
MOVL C01810 V=800.0 PL=0
MOVL C01811 V=800.0 PL=0
MOVL C01812 V=800.0 PL=0
MOVL C01813 V=800.0 PL=0
MOVL C01814 V=800.0 PL=0
MOVL C01815 V=800.0 PL=0
MOVL C01816 V=800.0 PL=0
MOVL C01817 V=800.0 PL=0
MOVL C01818 V=800.0 PL=0
MOVL C01819 V=800.0 PL=0
MOVL C01820 V=800.0 PL=0
MOVL C01821 V=800.0 PL=0
MOVL C01822 V=800.0 PL=0
MOVL C01823 V=800.0 PL=0
MOVL C01824 V=800.0 PL=0
MOVL C01825 V=800.0 PL=0
MOVL C01826 V=800.0 PL=0
MOVL C01827 V=800.0 PL=0
MOVL C01828 V=800.0 PL=0
MOVL C01829 V=800.0 PL=0
MOVL C01830 V=800.0 PL=0
MOVL C01831 V=800.0 PL=0
MOVL C01832 V=800.0 PL=0
MOVL C01833 V=800.0 PL=0
MOVL C01834 V=800.0 PL=0
MOVL C01835 V=800.0 PL=0
MOVL C01836 V=800.0 PL=0
MOVL C01837 V=800.0 PL=0
MOVL C01838 V=800.0 PL=0
MOVL C01839 V=800.0 PL=0
MOVL C01840 V=800.0 PL=0
MOVL C01841 V=800.0 PL=0
MOVL C01842 V=800.0 PL=0
MOVL C01843 V=800.0 PL=0
MOVL C01844 V=800.0 PL=0
MOVL C01845 V=800.0 PL=0
MOVL C01846 V=800.0 PL=0
MOVL C01847 V=800.0 PL=0
MOVL C01848 V=800.0 PL=0
MOVL C01849 V=800.0 PL=0
MOVL C01850 V=800.0 PL=0
MOVL C01851 V=800.0 PL=0
MOVL C01852 V=800.0 PL=0
MOVL C01853 V=800.0 PL=0
MOVL C01854 V=800.0 PL=0
MOVL C01855 V=800.0 PL=0
MOVL C01856 V=800.0 PL=0
MOVL C01857 V=800.0 PL=0
MOVL C01858 V=800.0 PL=0
MOVL C01859 V=800.0 PL=0
MOVL C01860 V=800.0 PL=0
MOVL C01861 V=800.0 PL=0
MOVL C01862 V=800.0 PL=0
MOVL C01863 V=800.0 PL=0
MOVL C01864 V=800.0 PL=0
MOVL C01865 V=800.0 PL=0
MOVL C01866 V=800.0 PL=0
MOVL C01867 V=800.0 PL=0
MOVL C01868 V=800.0 PL=0
MOVL C01869 V=800.0 PL=0
MOVL C01870 V=800.0 PL=0
MOVL C01871 V=800.0 PL=0
MOVL C01872 V=800.0 PL=0
MOVL C01873 V=800.0 PL=0
MOVL C01874 V=800.0 PL=0
MOVL C01875 V=800.0 PL=0
MOVL C01876 V=800.0 PL=0
MOVL C01877 V=800.0 PL=0
MOVL C01878 V=800.0 PL=0
MOVL C01879 V=800.0 PL=0
MOVL C01880 V=800.0 PL=0
MOVL C01881 V=800.0 PL=0
MOVL C01882 V=800.0 PL=0
MOVL C01883 V=800.0 PL=0
MOVL C01884 V=800.0 PL=0
MOVL C01885 V=800.0 PL=0
MOVL C01886 V=800.0 PL=0
MOVL C01887 V=800.0 PL=0
MOVL C01888 V=800.0 PL=0
MOVL C01889 V=800.0 PL=0
MOVL C01890 V=800.0 PL=0
MOVL C01891 V=800.0 PL=0
MOVL C01892 V=800.0 PL=0
MOVL C01893 V=800.0 PL=0
MOVL C01894 V=800.0 PL=0
MOVL C01895 V=800.0 PL=0
MOVL C01896 V=800.0 PL=0
MOVL C01897 V=800.0 PL=0
MOVL C01898 V=800.0 PL=0
MOVL C01899 V=800.0 PL=0
MOVL C01900 V=800.0 PL=0
MOVL C01901 V=800.0 PL=0
MOVL C01902 V=800.0 PL=0
MOVL C01903 V=800.0 PL=0
MOVL C01904 V=800.0 PL=0
MOVL C01905 V=800.0 PL=0
MOVL C01906 V=800.0 PL=0
MOVL C01907 V=800.0 PL=0
MOVL C01908 V=800.0 PL=0
MOVL C01909 V=800.0 PL=0
MOVL C01910 V=800.0 PL=0
MOVL C01911 V=800.0 PL=0
MOVL C01912 V=800.0 PL=0
MOVL C01913 V=800.0 PL=0
MOVL C01914 V=800.0 PL=0
MOVL C01915 V=800.0 PL=0
MOVL C01916 V=800.0 PL=0
MOVL C01917 V=800.0 PL=0
MOVL C01918 V=800.0 PL=0
MOVL C01919 V=800.0 PL=0
MOVL C01920 V=800.0 PL=0
MOVL C01921 V=800.0 PL=0
MOVL C01922 V=800.0 PL=0
MOVL C01923 V=800.0 PL=0
MOVL C01924 V=800.0 PL=0
MOVL C01925 V=800.0 PL=0
MOVL C01926 V=800.0 PL=0
MOVL C01927 V=800.0 PL=0
MOVL C01928 V=800.0 PL=0
MOVL C01929 V=800.0 PL=0
MOVL C01930 V=800.0 PL=0
MOVL C01931 V=800.0 PL=0
MOVL C01932 V=800.0 PL=0
MOVL C01933 V=800.0 PL=0
MOVL C01934 V=800.0 PL=0
MOVL C01935 V=800.0 PL=0
MOVL C01936 V=800.0 PL=0
MOVL C01937 V=800.0 PL=0
MOVL C01938 V=800.0 PL=0
MOVL C01939 V=800.0 PL=0
MOVL C01940 V=800.0 PL=0
MOVL C01941 V=800.0 PL=0
MOVL C01942 V=800.0 PL=0
MOVL C01943 V=800.0 PL=0
MOVL C01944 V=800.0 PL=0
MOVL C01945 V=800.0 PL=0
MOVL C01946 V=800.0 PL=0
MOVL C01947 V=800.0 PL=0
MOVL C01948 V=800.0 PL=0
MOVL C01949 V=800.0 PL=0
MOVL C01950 V=800.0 PL=0
MOVL C01951 V=800.0 PL=0
MOVL C01952 V=800.0 PL=0
MOVL C01953 V=800.0 PL=0
MOVL C01954 V=800.0 PL=0
MOVL C01955 V=800.0 PL=0
MOVL C01956 V=800.0 PL=0
MOVL C01957 V=800.0 PL=0
MOVL C01958 V=800.0 PL=0
MOVL C01959 V=800.0 PL=0
MOVL C01960 V=800.0 PL=0
MOVL C01961 V=800.0 PL=0
MOVL C01962 V=800.0 PL=0
MOVL C01963 V=800.0 PL=0
MOVL C01964 V=800.0 PL=0
MOVL C01965 V=800.0 PL=0
MOVL C01966 V=800.0 PL=0
MOVL C01967 V=800.0 PL=0
MOVL C01968 V=800.0 PL=0
MOVL C01969 V=800.0 PL=0
MOVL C01970 V=800.0 PL=0
MOVL C01971 V=800.0 PL=0
MOVL C01972 V=800.0 PL=0
MOVL C01973 V=800.0 PL=0
MOVL C01974 V=800.0 PL=0
MOVL C01975 V=800.0 PL=0
MOVL C01976 V=800.0 PL=0
MOVL C01977 V=800.0 PL=0
MOVL C01978 V=800.0 PL=0
MOVL C01979 V=800.0 PL=0
MOVL C01980 V=800.0 PL=0
MOVL C01981 V=800.0 PL=0
MOVL C01982 V=800.0 PL=0
MOVL C01983 V=800.0 PL=0
MOVL C01984 V=800.0 PL=0
MOVL C01985 V=800.0 PL=0
MOVL C01986 V=800.0 PL=0
MOVL C01987 V=800.0 PL=0
MOVL C01988 V=800.0 PL=0
MOVL C01989 V=800.0 PL=0
MOVL C01990 V=800.0 PL=0
MOVL C01991 V=800.0 PL=0
MOVL C01992 V=800.0 PL=0
MOVL C01993 V=800.0 PL=0
MOVL C01994 V=800.0 PL=0
MOVL C01995 V=800.0 PL=0
MOVL C01996 V=800.0 PL=0
MOVL C01997 V=800.0 PL=0
MOVL C01998 V=800.0 PL=0
MOVL C01999 V=800.0 PL=0
MOVL C02000 V=800.0 PL=0
MOVL C02001 V=800.0 PL=0
MOVL C02002 V=800.0 PL=0
MOVL C02003 V=800.0 PL=0
MOVL C02004 V=800.0 PL=0
MOVL C02005 V=800.0 PL=0
MOVL C02006 V=800.0 PL=0
MOVL C02007 V=800.0 PL=0
MOVL C02008 V=800.0 PL=0
MOVL C02009 V=800.0 PL=0
MOVL C02010 V=800.0 PL=0
MOVL C02011 V=800.0 PL=0
MOVL C02012 V=800.0 PL=0
MOVL C02013 V=800.0 PL=0
MOVL C02014 V=800.0 PL=0
MOVL C02015 V=800.0 PL=0
MOVL C02016 V=800.0 PL=0
MOVL C02017 V=800.0 PL=0
MOVL C02018 V=800.0 PL=0
